activate_last := ACTIVATE; (* letzten Status sichern zur Flankenerkennung *)

(* IP_FIFO *)
IP_FIFO(FIFO:=IP_C.FIFO,STATE:=ip_state,ID:=ip_id);

(* revision history
ks	18. oct. 2008	rev 1.0
	original version

ks	20. oct. 2009	rev 1.1
	Networkbuffer und Buffer-funktionen auf Basis 0

*)

(***************************************************************************************)
(*               SNTP Datenstruktur
                                  1                   2                   3   
              0 1 2 3 4 5 6 7 8 9 0 1 2 3 4 5 6 7 8 9 0 1 2 3 4 5 6 7 8 9 0 1 
             +-+-+-+-+-+-+-+-+-+-+-+-+-+-+-+-+-+-+-+-+-+-+-+-+-+-+-+-+-+-+-+-+
Byte: 01-04  |LI | VN  |Mode |    Stratum    |     Poll      |   Precision   |
             +-+-+-+-+-+-+-+-+-+-+-+-+-+-+-+-+-+-+-+-+-+-+-+-+-+-+-+-+-+-+-+-+
Byte: 05-08  |                          Root  Delay (32 Bit)                 |
             +-+-+-+-+-+-+-+-+-+-+-+-+-+-+-+-+-+-+-+-+-+-+-+-+-+-+-+-+-+-+-+-+
Byte: 09-12  |                       Root  Dispersion (32 Bit)               |
             +-+-+-+-+-+-+-+-+-+-+-+-+-+-+-+-+-+-+-+-+-+-+-+-+-+-+-+-+-+-+-+-+
Byte: 13-16  |                     Reference Identifier (32 Bit)             |
             +-+-+-+-+-+-+-+-+-+-+-+-+-+-+-+-+-+-+-+-+-+-+-+-+-+-+-+-+-+-+-+-+
Byte: 17-24  |                    Reference Timestamp (64 Bit)               |
             +-+-+-+-+-+-+-+-+-+-+-+-+-+-+-+-+-+-+-+-+-+-+-+-+-+-+-+-+-+-+-+-+
Byte: 25-32  |                    Originate Timestamp (64 Bit)               |
             +-+-+-+-+-+-+-+-+-+-+-+-+-+-+-+-+-+-+-+-+-+-+-+-+-+-+-+-+-+-+-+-+
Byte: 33-40  |                     Receive Timestamp (64 Bit)                |
             +-+-+-+-+-+-+-+-+-+-+-+-+-+-+-+-+-+-+-+-+-+-+-+-+-+-+-+-+-+-+-+-+
Byte: 41-48  |                     Transmit Timestamp (64 Bit)               |
             +-+-+-+-+-+-+-+-+-+-+-+-+-+-+-+-+-+-+-+-+-+-+-+-+-+-+-+-+-+-+-+-+
Byte: 49-52  |                 Key Identifier (optional) (32 Bit)            |
             +-+-+-+-+-+-+-+-+-+-+-+-+-+-+-+-+-+-+-+-+-+-+-+-+-+-+-+-+-+-+-+-+
Byte: 53-68  |                 Message Digest (optional) (128 Bit)           |
             +-+-+-+-+-+-+-+-+-+-+-+-+-+-+-+-+-+-+-+-+-+-+-+-+-+-+-+-+-+-+-+-+

*)

(*
Worldwide NTP-Server


NIST-Zeitserver
• time-a.nist.gov
129.6.15.28 
NIST, Gaithersburg, Maryland 
• time-a.nist.gov
129.6.15.28 
NIST, Gaithersburg, Maryland 
• time-a.timefreq.bldrdoc.gov
132.163.4.101 (Stand: 1. Dezember 1999)
NIST, Boulder, Colorado 
• time-b.timefreq.bldrdoc.gov
132.163.4.102 (Stand: 1. Dezember 1999)
NIST, Boulder, Colorado 
• time-c.timefreq.bldrdoc.gov
132.163.4.103 (Stand: 1. Dezember 1999)
NIST, Boulder, Colorado 
• utcnist.colorado.edu
128.138.140.44
University of Colorado, Boulder 
• time.nist.gov
192.43.244.18
NCAR, Boulder, Colorado 
• time-nw.nist.gov
131.107.1.10
Microsoft, Redmond, Washington 
• nist1.dc.certifiedtime.com
216.200.93.8
Abovnet, North Virginia 
• nist1.datum.com
209.0.72.7
Datum, San Jose, Kalifornien 
• nist1.nyc.certifiedtime.com
208.184.49.129 
Abovnet, New York City 
• nist1.sjc.certifiedtime.com
207.126.103.202
Abovnet, San Jose, Kalifornien 

Zeitserver der ersten Ebene
Sortiert nach Standort: 
Nordamerika
• Palo Alto, Kalifornien: Systems Research Center, Compaq Computer Corp.
204.123.2.72: usno.pa-x.dec.com; CNAME: navobs1.pa-x.dec.com
Servicebereich: US-Zeitzonen PST (Pacific Standard Time) und MST (Mountain Standard Time) 
• Marina del Rey, Kalifornien: USC Information Sciences Institute
128.9.176.30: timekeeper.isi.edu
Servicebereich: CalRen2- und Los Nettos-Bereich  
• Washington, DC: U.S. Naval Observatory
192.5.41.41: tock.usno.navy.mil 
192.5.41.40: tick.usno.navy.mil
Servicebereich: NSFNET 
• Ottawa, Ontario, Kanada: National Research Council of Canada
time.chu.nrc.ca
Servicebereich: Kanada 
• Raleigh, North Carolina: North Carolina State University
152.1.58.124: terrapin.csc.ncsu.edu
Servicebereich: Südosten der USA 
• Cambridge, Massachusetts: MIT Information Systems
18.72.0.3: bitsy.mit.edu 
Servicebereich: NSFNET- und NEARnet-Bereich 
• Cambridge, Massachusetts: MIT
18.26.4.105: bonehed.lcs.mit.edu
Servicebereich: Osten der USA 
• Palo Alto, Kalifornien: Internet Software Consortium
192.5.5.250: clock.isc.org
Servicebereich: BARRnet, Alternet-West und CIX-West 
• Cambridge, Massachusetts: Open Software Foundation
130.105.4.59: clock.osf.org
Servicebereich: NSFNET- und NEARnet-Bereich 
• Palo Alto, Kalifornien: ViaNet Communications
209.81.9.7: clock.via.net 
• Cleveland, Ohio: Lewis Research Center (NASA)
128.156.1.43: lerc-dns.lerc.nasa.gov
Servicebereich: NSFNET und OARNET 
• Colorado Springs, Colorado: Schriever AFB
204.34.198.40: navobs1.usnogps.navy.mil; CNAME: tick.usnogps.navy.mil 
204.34.198.41: navobs1.usnogps.navy.mil; CNAME: tock.usnogps.navy.mil 
Servicebereich: US-Zeitzonen PST (Pacific Standard Time) und MST (Mountain Standard Time) 
• St. Louis, Missouri: Washington University
128.252.19.1: navobs1.usnogps.navy.mil; CNAME: tick.wustl.edu 
Servicebereich: US-Zeitzone CST (Central Standard Time) 
• Research Triangle Park, North Carolina: MCNC
192.101.21.1: ncnoc.ncren.net
Servicebereich: NC-REN-Bereich (North Carolina Research and Education Network) 
• Cupertino, Kalifornien: HP
192.6.38.127: ntp-cup.external.hp.com
Servicebereich: USA Westküste 
• Newark, Delaware: Conectiv Communications
138.39.7.20: ntp1.delmarva.com
Servicebereich: Cable & Wireless Network (früher MCInet) 
• University Park, Pennsylvania: Penn State University
128.118.46.3: otc1.psu.edu
Servicebereich: NSFNET, PREPNET und JvNCnet  

Europa
• Borowiec, Polen: Astrogeodynamical Observatory, Space Research Centre
150.254.183.15: vega.cbk.poznan.pl
Servicebereich: Polen und Europa 
• Stockholm, Schweden: Stupi AB
192.36.143.151: Time2.Stupi.SE
Servicebereich: Europa 
• Turin, Italien: IEN Galileo Ferraris
193.204.114.1: time.ien.it
Servicebereich: Italien und Europa 
• Zürich, Schweiz: Integrated Systems Laboratory , Eidgenössischen Technischen Hochschule Zürich 
129.132.2.21: swisstime.ethz.ch
Servicebereich: Schweiz und Europa 
• Turin, Italien: CSTV of National Research Council
150.145.33.1: tempo.cstv.to.cnr.it
Servicebereich: Italien und Europa 
• Erlangen, Deutschland: Universität Erlangen-Nürnberg
ntp0.fau.de; ntp1.fau.de; ntp2.fau.de; 
ntps1-0.uni-erlangen.de; ntps1-1.uni-erlangen.de; ntps1-2.uni-erlangen.de
Servicebereich: Deutschland und Europa 
• Berlin, Deutschland: Technische Universität Berlin
130.149.17.21: ntps1-0.cs.tu-berlin.de
130.149.17.8: ntps1-1.cs.tu-berlin.de
Servicebereich: Deutschland und Europa 
• Deutschland
131.173.17.7: ntps1-1.rz.Uni-Osnabrueck.DE
Servicebereich: Deutschland und Europa 
• Schweden
192.36.143.150: Time1.Stupi.SE
Servicebereich: SUnet und NORDUnet Schweden 

Fernost und pazifische Randgebiete
• Hong Kong: Chinesische Universität von Hong Kong. 
137.189.6.18: clock.cuhk.edu.hk
Servicebereich: Hong Kong (China) und Südostasien  
• Fukuoka, Japan: Universität Fukuoka
133.100.9.2: clock.nc.fukuoka-u.ac.jp
133.100.11.8: clock.tl.fukuoka-u.ac.jp
Servicebereich: Japan und pazifischer Raum  

Australien
• Melbourne, Australien: University of Melbourne
128.250.36.2: ntp.cs.mu.OZ.AU
Servicebereich: Australien und Neuseeland  

Zeitserver der zweiten Ebene
Nach geographischem Standort sortiert: 
Nordamerika
NTP-Zeitserver: • Quebec, Kanada: Canadian Meteorological Center
ntp1.cmc.ec.gc.ca; ntp2.cmc.ec.gc.ca 
Servicebereich: Ostkanada  
• Ontario, Kanada: National Research Council of Canada
time.chu.nrc.ca; time.nrc.ca
Servicebereich: Kanada 
• Saskatchewan, Kanada: University of Regina 
142.3.100.15: timelord.uregina.ca
Servicebereich: Kanada 
• Ontario, Kanada: University of Toronto
tick.utoronto.ca; tock.utoronto.ca
Servicebereich: Ostkanada  
• Mexiko: Audiotel-Büro 
ntp2a.audiotel.com.mx; ntp2c.audiotel.com.mx; ntp2b.audiotel.com.mx
Servicebereich: Avantel, MCINet und Mexiko 
• Santa Cruz, Kalifornien: Scruz-net, inc.
165.227.1.1: ns.scruz.net
Servicebereich: Westen der USA 
• San Diego, Kalifornien: UCSD Academic Computing Services/Network Operations
132.239.254.49: ntp.ucsd.edu
Servicebereich: CERFNET; NSFNET, SDSC-Bereich, und nahegelegene Bereiche 
• Quincy, Kalifornien 
ntp1.mainecoon.com; ntp2.mainecoon.com 
Servicebereich: Nordamerika 
• Newark, Delaware: University of Delaware
128.175.1.3: louie.udel.edu
Servicebereich: CAIRN, Abilene und vBNS  
• Atlanta, Georgia: CNSG
ntp.shorty.com
Servicebereich: Südwesten der USA  
• Kennesaw, Georgia: PeachNet 
rolex.peachnet.edu; timex.peachnet.edu
Servicebereich: PeachNet (Georgia) und Südwesten der USA  
• Urbana-Champaign, Illinois: University of Illinois
ntp-0.cso.uiuc.edu; ntp-1.cso.uiuc.edu; ntp-2.cso.uiuc.edu
Servicebereich: CICNET, Mittlerer Westen und NCSA-Bereich  
• Chicago, Illinois: Argonne National Laboratory 
ntp-1.mcs.anl.gov; ntp-2.mcs.anl.gov
Servicebereich: NSF/ANSNet, CICNet, NetIllinois und ESNet  
• West Lafayette, Indiana: Purdue University
gilbreth.ecn.purdue.edu; harbor.ecn.purdue.edu; molecule.ecn.purdue.edu 
Servicebereich: NSFNET- und CICNET-Bereich  
• Manhattan, Kansas: KansasNet OnLine Services
199.240.130.1: ntp1.kansas.net
199.240.130.12: ntp2.kansas.net
Servicebereich: Zentral-USA und Great Plains  
• Boston, Massachusetts: UMass-Boston CS dept.
158.121.104.4: timeserver.cs.umb.edu
Servicebereich: Neuengland  
• Minneapolis/St Paul, Minnesota: University of Minnesota
ns.nts.umn.edu; nss.nts.umn.edu
Servicebereich: CICNET-Bereich  
• Columbia, Missouri: University of Missouri-Columbia
128.206.206.12: everest.cclabs.missouri.edu
Servicebereich: MOREnet  
• Omaha, Nebraska: Radiks Internet Access
205.138.126.83: allison.radiks.net
Servicebereich: Mittlerer Westen, USA  
• Las Vegas, Nevada: University of Nevada System Computing Services
131.216.1.101: cuckoo.nevada.edu 
Servicebereich: NevadaNet, NSFNET und SDSC-Bereich  
• Las Vegas, Nevada: UNLV College of Engineering
tick.cs.unlv.edu; tock.cs.unlv.edu
Servicebereich: Sprintnet  
• New York City, New York: Columbia University
ntp.ctr.columbia.edu 
Servicebereich: Sprintlink und NYSERnet  
• Ithaca, New York: Cornell University 
192.35.82.50: ntp0.cornell.edu
Servicebereich: NSFNET und NYSER-Bereich  
• New York, New York: Morningside Campus, Columbia University
sundial.columbia.edu
Servicebereich: NYSERnet  
• New York City, New York: Columbia University Computer Science Department
timex.cs.columbia.edu 
Servicebereich: PSINET; NSFNET, und NYSER-Bereich  
• Norman, Oklahoma: University of Oklahoma
129.15.22.8: constellation.ecn.uoknor.edu 
Servicebereich: Midnet  
• Coos Bay, Oregon: Koala Computers
207.48.109.6: tick.koalas.com
Servicebereich: Nordwesten der USA  
• University Park, Pennsylvania: Penn State University
128.118.25.3: clock.psu.edu
Servicebereich: Internet2, vBNS, CERFnet(AT&T IP Services), PSC/NCNE und CASC 
• Pittsburgh, Pennsylvania: Pittsburgh Supercomputing Center
128.182.58.100: fuzz.psc.edu
Servicebereich: NSFNET und PSC-Bereich  
• Pittsburgh, Pennsylvania: Carnegie Mellon Electrical and Computer Engineering 
ntp-1.ece.cmu.edu; ntp-2.ece.cmu.edu 
Servicebereich: PREPNET und PSC-Bereich  
• Dallas, Texas: Cox School of Business, Southern Methodist University
129.119.80.126: ntp.cox.smu.edu 
Servicebereich: NSFNET und SESQUI-Bereich  
• Hughes Springs, Texas: First National Bank
209.144.20.76: ntp.fnbhs.com
Servicebereich: Nordosten Texas  
• Houston, Texas: Baylor College of Medicine
128.249.1.10: ntp.tmc.edu 
Servicebereich: NSFNET und SESQUI-Bereich  
• College Station, Texas: Texas A&M University
165.91.52.110: ntp5.tamu.edu
Servicebereich: NSFNET, SESQUI-Bereich, THEnet und TAMUSDSN 
• Plano, Texas: Greyware Automation Products
tick.greyware.com; tock.greyware.com
Servicebereich: Südzentral-USA  
• Blacksburg, Virginia: Virginia Tech Computing Center
ntp-1.vt.edu; ntp-2.vt.edu
Servicebereich: Südwesten der USA  
• Arlington, Virginia: Center for Seismic Studies
140.162.1.3: ntp.cmr.gov
Servicebereich: NSFNET und SURA-Bereich  
• Richland, Washington: Washington State University 
192.31.216.30: clock.tricity.wsu.edu
Servicebereich: NSFNET und NorthWestNet  
• Washington, USA: Mill Creek
time.ultimeth.net
Servicebereich: Nordwesten der USA  
• Wisconsin, USA: Computer Science Department, University of Wisconsin-Madison
ntp1.cs.wisc.edu; ntp2.cs.wisc.edu; ntp3.cs.wisc.edu
Servicebereich: USA und jeder andere  

Südamerika
• Buenos Aires, Argentinien: Network Access Point
200.49.40.1: CNAME: tick.nap.com.ar
200.49.32.1: CNAME: tock.nap.com.ar
Servicebereich: Argentinien 
• Buenos Aires, Argentinien: Sinectis S.A.
time.sinectis.com.ar 
Servicebereich: Argentinien 
• Brasilien: Brazilian Research Network
200.144.121.33: ntp.cais.rnp.br 
Servicebereich: Brasilien 
• Venezuela: VELUG, Grupo de Usuarios Linux de Venezuela
150.185.192.250: ntp.linux.org.ve
Servicebereich: Arica  

Europa
• Zürich, Schweiz: Eidgenössischen Technischen Hochschule Zürich
129.132.98.11: bernina.ethz.ch
Servicebereich: Schweiz und Europa  
• Standort: Kopenhagen, Dänemark, Europa 
clock.netcetera.dk; clock2.netcetera.dk 
Servicebereich: Dänemark, Skandinavien und Nordeuropa  
• Spanien: Altea 
slug.ctv.es
Servicebereich: Spanien  
• Pieksamaki, Finnland: Keski-Savon Oppimiskeskus
tick.keso.fi; tock.keso.fi
Servicebereich: Finnland  
• Meudon, Frankreich: Observatoire de Paris-Meudon 
ntp.obspm.fr 
Servicebereich: Frankreich und Europa  
• Lyon, Frankreich: CISM 
ntp.univ-lyon1.fr 
Servicebereich: Frankreich, Schweiz, Italien und Europa  
• Paris, Frankreich: VIA, Ecole Centrale
138.195.130.70: ntp.via.ecp.fr
Servicebereich: Frankreich und Europa  
• Budapest, Ungarn: KFKI Research Institute for Particle and Nuclear Physics
148.6.0.1: time.kfki.hu
Servicebereich: HUNGARNET  
• Italien: Net4u Srl, Vercelli, Italien
195.32.52.129: ntps.net4u.it
Servicebereich: Italien  
• Oslo, Norwegen: Universität Oslo
129.240.64.3: fartein.ifi.uio.no 
Servicebereich: NORDUnet  
• Oslo, Norwegen: Alcanet International
time.alcanet.no
Servicebereich: Europa 
• Krakau, Polen: Academic Computer Centre 
149.156.4.11: info.cyf-kr.edu.pl
Servicebereich: Polen und Europa  
• Lund, Schweden: Lund Institute of Technology
130.235.20.3: ntp.lth.se 
Servicebereich: Schweden und NORDUnet 
• Ljubljana, Slowenien: Institute of Biophysics, University of Ljubljana
biofiz.mf.uni-lj.si 193.2.69.11
Servicebereich: Slowenien und Europa  
• Ljubljana, Slowenien: Hydrometeorological Institute of Slovenia
hmljhp.rzs-hm.si
Servicebereich: Slowenien und Europa  
• Ljubljana, Slowenien: Academic and Research Network of Slovenia
ntp1.arnes.si; ntp2.arnes.si
Servicebereich: Slowenien und Europa  
• Ljubljana, Slowenien: J. Stefan Institute
time.ijs.si
Servicebereich: Slowenien und Europa  

Britische Inseln
• Dublin, Irland: School of Mathematics, Trinity College 
ntp.cs.tcd.ie; ntp.maths.tcd.ie; ntp.tcd.ie
Servicebereich: Irland und Großbritannien 
• Glasgow, Schottland: Strathclyde University 
ntp.cs.strath.ac.uk 
Servicebereich: Großbritannien, Europa und andere 
• Cambridge, Großbritannien
ntp0.uk.uu.net; ntp1.uk.uu.net; 
ntp2.uk.uu.net 
Servicebereich: UUNET (in Großbritannien früher auch als PIPEX bekannt) und Großbritannien.  
• Manchester, England: University of Manchester
ntp2a.mcc.ac.uk; ntp2b.mcc.ac.uk;
ntp2c.mcc.ac.uk; ntp2d.mcc.ac.uk 
Servicebereich: Großbritannien  
• Buckinghamshire, Großbritannien: Wibble U.K., Aylesbury
tick.tanac.net
Servicebereich: Großbritannien  

Asien
• Moskau, Russland: Landau Institute for Theoretical Physics
193.233.9.7: ntp.landau.ac.ru
Servicebereich: Russland  
• Russland: Pushchino (bei Moskau)
194.149.67.130: ntp.psn.ru
Servicebereich: Russland 
• Chernogolovka, Russland: Chernogolovka Scientific Center (bei Moskau)
193.233.46.10: sign.chg.ru
Servicebereich: Russland  

Fernost und pazifische Randgebiete
• Tokyo, Japan: Cyber Fleet, Inc.
203.139.30.195: ntp.cyber-fleet.net
Servicebereich: Japan und Ostasien  
• Seoul, Korea: Inet, Inc.
time.nuri.net
Servicebereich: Korea, Japan, Hong Kong und Ostasien  
• Hamilton, Neuseeland: Universität Waikato
truechimer.waikato.ac.nz; truechimer1.waikato.ac.nz; 
truechimer2.waikato.ac.nz; truechimer3.waikato.ac.nz
Servicebereich: Neuseeland  
• Singapur und Philippinen: 
ntp.shim.org 
Servicebereich: Singapur  

Afrika
• Lagos, Nigeria: Supernet300
ntp.supernet300.com
Servicebereich: Westafrika (hauptsächlich nigerischer NITEL-Backbone)  
• Pietermaritzburg, Südafrika: Natal University
143.128.82.200: ntp.cs.unp.ac.za
Servicebereich: Südafrika  

Australien
• Adelaide, Südaustralien: University of Adelaide
129.127.28.4: augean.eleceng.adelaide.edu.au
129.127.40.3: ntp.adelaide.edu.au
203.21.37.18: ntp.saard.net
Servicebereich: AARNet  
• Carlton, Victoria, Australien: eSec Limited
203.21.84.4: time.esec.com.au  

*)
END_FUNCTION_BLOCK

(* POU SNTP_SERVER, ST *)
FUNCTION_BLOCK SNTP_SERVER
VAR_IN_OUT
	IP_C : IP_C; (* IP_Control Verwaltungsstruktur *)
	S_BUF : NETWORK_BUFFER;
	R_BUF : NETWORK_BUFFER;
END_VAR
VAR_INPUT
	ENABLE : BOOL;
	STRATUM : BYTE := BYTE#1;
	UDT : DT;
	XMS : INT;
END_VAR
VAR
	IP_FIFO : IP_FIFO;
	ip_state : BYTE;
	ip_id : BYTE;
	i2 : INT;
	i : INT;
	timestamp_int : DWORD; (* Timestamp integer part *)
	timestamp_sek : DWORD; (* Timestamp fraction part (HIGH_WORD) *)
	ts_b : BYTE;
	state : INT;
	tx : UDINT;
END_VAR

(*
	version 1.1		20. oct. 2009
	programmer 		ks
	tested BY		ks

	SNTP_SERVER stellt Datum/Uhrzeit füR andere (S)NTP_CLIENTS zur Verfügung.
*)
(* Domain Name System (query) *)
tx := T_PLC_MS(); (* read system time *)

CASE state OF

00: (* Warten auf Freigabe *)
	IF ENABLE THEN
		state := 10;
		ip_state := BYTE#1; (* Anmelden *)
	END_IF;

10: (* Bei IP_Control anmelden und auf freigabe warten *)
	IF ip_state = BYTE#3 THEN
		(* IP Datenverkehr einrichten *)
		IP_C.C_PORT := WORD#123; (* Portnummer eintragen *)
		IP_C.C_IP := DWORD#00; (* IP eintragen *)
		IP_C.C_MODE := BYTE#5; (* Mode: UDP+PASSIV+PORT *)
		IP_C.C_ENABLE := TRUE; (* Verbindungsaufbau freigeben *)
		IP_C.TIME_RESET := TRUE; (* Zeitueberwachung rücksetzen *)
		IP_C.R_OBSERVE := FALSE; (* Datenempfang ueberwachen *)
		S_BUF.SIZE := UINT#0; (* Sendelänge eintragen *)
		R_BUF.SIZE := UINT#0; (* Empfangslänge rücksetzen *)
		state := 20;
	END_IF;
20:
	IF R_BUF.SIZE > UINT#0 THEN
		state := 20;
		(* empfangenes Telegramm mit 00 auffüllen , wenn zu kurz ! und Sendebuffer mit 00 vorbelegen *)
		FOR i := 0 TO 47 DO
			IF INT_TO_UINT(i) > R_BUF.SIZE - 1 THEN
				R_BUF.BUFFER[i] := BYTE#00;
			END_IF;
			S_BUF.BUFFER[i] := BYTE#00;
		END_FOR;

		R_BUF.SIZE := UINT#0;

		(* Sendedaten aufbereiten *)
		S_BUF.BUFFER[0] := BYTE#2#11100; (* Flags: NO WARNING, NTP VERSION 3 , SERVER *)
		S_BUF.BUFFER[1] := STRATUM; (* Peer Clock Stratum: *)
		S_BUF.BUFFER[2] := BYTE#10; (* Peer Polling Intervall 2 hoch 10 = 1024 sek. *)
		S_BUF.BUFFER[3] := BYTE#16#FB; (* Peer Clock Precision: -5 = -31,25ms *)

		(* Umrechnung SNTP Timestamp Base 1900-01-01 = Unix 1970-01-01 + 2208988800 sekunden *)
		timestamp_int := DT_TO_DWORD(UDT) + DWORD#2208988800;

		(* Sekundenanteile sind als 32 Bit Fractal dargestellt *)
		(* nur mit veringerte Auflösung berechnen 1/65535 -> Highword verwenden *)
		(* Berechnung des Sekundenanteils: xms * 65535 / 1000 *)
		timestamp_sek := DINT_TO_DWORD(DWORD_TO_DINT(SHL(INT_TO_DWORD(XMS),16))/DINT#1000);

		ts_b := BYTE_OF_DWORD(timestamp_int,3); (* Timestamp Byte 3 *)
		S_BUF.BUFFER[16] := ts_b; (* Reference Timestamp *)
		S_BUF.BUFFER[32] := ts_b; (* Receive   Timestamp *)
		S_BUF.BUFFER[40] := ts_b; (* Transmit  Timestamp *)

		ts_b := BYTE_OF_DWORD(TIMESTAMP_INT,2); (* Timestamp Byte 2 *)
		S_BUF.BUFFER[17] := ts_b; (* Reference Timestamp *)
		S_BUF.BUFFER[33] := ts_b; (* Receive   Timestamp *)
		S_BUF.BUFFER[41] := ts_b; (* Transmit  Timestamp *)

		ts_b := BYTE_OF_DWORD(TIMESTAMP_INT,1); (* Timestamp Byte 1 *)
		S_BUF.BUFFER[18] := ts_b; (* Reference Timestamp *)
		S_BUF.BUFFER[34] := ts_b; (* Receive   Timestamp *)
		S_BUF.BUFFER[42] := ts_b; (* Transmit  Timestamp *)

		ts_b := BYTE_OF_DWORD(TIMESTAMP_INT,0); (* Timestamp Byte 0 *)
		S_BUF.BUFFER[19] := ts_b; (* Reference Timestamp *)
		S_BUF.BUFFER[35] := ts_b; (* Receive   Timestamp *)
		S_BUF.BUFFER[43] := ts_b; (* Transmit  Timestamp *)

		ts_b := BYTE_OF_DWORD(TIMESTAMP_SEK,1); (* Timestamp Byte 1 *)
		S_BUF.BUFFER[20] := ts_b; (* Reference Timestamp *)
		S_BUF.BUFFER[36] := ts_b; (* Receive   Timestamp *)
		S_BUF.BUFFER[44] := ts_b; (* Transmit  Timestamp *)

		ts_b := BYTE_OF_DWORD(timestamp_sek,0);	(* Timestamp Byte 0 *)
		S_BUF.BUFFER[21] := ts_b; (* Reference Timestamp *)
		S_BUF.BUFFER[37] := ts_b; (* Receive   Timestamp *)
		S_BUF.BUFFER[45] := ts_b; (* Transmit  Timestamp *)

		(* Byte 1-8 von Transmit-Time auf Originate-Time umkopieren *)
		i2 := 40;
		FOR i := 24 TO 31 DO
			S_BUF.BUFFER[i] := R_BUF.BUFFER[i2];
			i2 := i2 +1;
		END_FOR;

		S_BUF.SIZE := UINT#48; (* Daten senden *)

	ELSIF NOT ENABLE AND S_BUF.SIZE = UINT#0 THEN
		ip_state := BYTE#4; (* Abmelden *)
		state := 0;
	END_IF;

END_CASE;

(* IP_FIFO *)
IP_FIFO(FIFO:=IP_C.FIFO,STATE:=ip_state,ID:=ip_id);

(* revision history
ks	18. oct. 2008	rev 1.0
	original version

ks	20. oct. 2009	rev 1.1
	Networkbuffer und Buffer-funktionen auf Basis 0

*)


(*               SNTP(NTP) Datenstruktur
                                  1                   2                   3
              0 1 2 3 4 5 6 7 8 9 0 1 2 3 4 5 6 7 8 9 0 1 2 3 4 5 6 7 8 9 0 1
             +-+-+-+-+-+-+-+-+-+-+-+-+-+-+-+-+-+-+-+-+-+-+-+-+-+-+-+-+-+-+-+-+
Byte: 01-04  |LI | VN  |Mode |    Stratum    |     Poll      |   Precision   |
             +-+-+-+-+-+-+-+-+-+-+-+-+-+-+-+-+-+-+-+-+-+-+-+-+-+-+-+-+-+-+-+-+
Byte: 05-08  |                          Root  Delay (32 Bit)                 |
             +-+-+-+-+-+-+-+-+-+-+-+-+-+-+-+-+-+-+-+-+-+-+-+-+-+-+-+-+-+-+-+-+
Byte: 09-12  |                       Root  Dispersion (32 Bit)               |
             +-+-+-+-+-+-+-+-+-+-+-+-+-+-+-+-+-+-+-+-+-+-+-+-+-+-+-+-+-+-+-+-+
Byte: 13-16  |                     Reference Identifier (32 Bit)             |
             +-+-+-+-+-+-+-+-+-+-+-+-+-+-+-+-+-+-+-+-+-+-+-+-+-+-+-+-+-+-+-+-+
Byte: 17-24  |                    Reference Timestamp (64 Bit)               |
             +-+-+-+-+-+-+-+-+-+-+-+-+-+-+-+-+-+-+-+-+-+-+-+-+-+-+-+-+-+-+-+-+
Byte: 25-32  |                    Originate Timestamp (64 Bit)               |
             +-+-+-+-+-+-+-+-+-+-+-+-+-+-+-+-+-+-+-+-+-+-+-+-+-+-+-+-+-+-+-+-+
Byte: 33-40  |                     Receive Timestamp (64 Bit)                |
             +-+-+-+-+-+-+-+-+-+-+-+-+-+-+-+-+-+-+-+-+-+-+-+-+-+-+-+-+-+-+-+-+
Byte: 41-48  |                     Transmit Timestamp (64 Bit)               |
             +-+-+-+-+-+-+-+-+-+-+-+-+-+-+-+-+-+-+-+-+-+-+-+-+-+-+-+-+-+-+-+-+
Byte: 49-52  |                 Key Identifier (optional) (32 Bit)            |
             +-+-+-+-+-+-+-+-+-+-+-+-+-+-+-+-+-+-+-+-+-+-+-+-+-+-+-+-+-+-+-+-+
Byte: 53-68  |                 Message Digest (optional) (128 Bit)           |
             +-+-+-+-+-+-+-+-+-+-+-+-+-+-+-+-+-+-+-+-+-+-+-+-+-+-+-+-+-+-+-+-+
*)
END_FUNCTION_BLOCK

(* POU SYS_LOG, ST *)
FUNCTION_BLOCK SYS_LOG
VAR_IN_OUT
	IP_C : IP_C; (* IP_Control Verwaltungsstruktur *)
	S_BUF : NETWORK_BUFFER;
	R_BUF : NETWORK_BUFFER;
END_VAR
VAR_INPUT
	ACTIVATE : BOOL;
	LDT : DT;
	SERVER_IP4 : DWORD;
	PORT : WORD;
	FACILITY : BYTE;
	SEVERITY : BYTE;
	TAG : STRING(32);
	HOSTNAME : STRING;
	MESSAGE : STRING(STRING_LENGTH);
	OPTION : BYTE;
END_VAR
VAR_OUTPUT
	DONE_P : BOOL;
	ERROR : DWORD;
END_VAR
VAR
	ip_state : BYTE;
	ip_id : BYTE;
	IP_FIFO : IP_FIFO;
	activate_last : BOOL;
	state : INT;
	s1 : STRING(20);
	i : INT;
END_VAR

(*
version 1.1		20. jun. 2009
programmer 		ks
tested by		ks

SYSLOG versendet Meldungen auf Basis des SYSLOG-Standards

*)
CASE state OF
00: (* auf positive Flanke SET warten *)
	IF ACTIVATE AND NOT ACTIVATE_LAST THEN
		state := 10;
		ERROR := DWORD#0;
		IP_STATE := BYTE#1; (* Anmelden *)
	END_IF;
	DONE_P := FALSE;

10: (* Bei IP_Control anmelden und auf freigabe warten *)
	IF IP_STATE = BYTE#3 THEN
		(* Sendedaten aufbereiten *)
		i := 0;
		IF (OPTION AND BYTE#0000_0001) = BYTE#00 THEN (* Option: no priority Code *)
			(* Priority:  '<xx>' als dezimalwert *)
			(* BYTE: xxxx x...  = Facility *)
			(*       .... .xxx  = Level *)
			s1 := REPLACE('<P>',BYTE_TO_STRING(SHL(FACILITY,3) OR (SEVERITY AND BYTE#0000_0111)),1,2);
		ELSE
			s1 := '';
		END_IF;

		IF (OPTION AND BYTE#0000_0010) = BYTE#00 THEN (* Option: No Use Syslog RFC Header *)
			(* 'month day hh:mm:ss ' *)
			s1 := CONCAT(s1,DT_TO_STRF(DTI:=LDT,MS:=0,FMT:='#E #W #N:#R:#T ',LANG:=1));
			_STRING_TO_BUFFER(STR:=s1,POS:=i,PT:=ADR(S_BUF.BUFFER),SIZE:=UINT#1024);
			i := i + LEN(s1);
			(* ' sourcename eintragen *)
			_STRING_TO_BUFFER(STR:=HOSTNAME,POS:=i,PT:=ADR(S_BUF.BUFFER),SIZE:=UINT#1024);
			i := i + LEN(HOSTNAME);
			S_BUF.BUFFER[i] := BYTE#32; (* leerzeichen einfuegen *)
			i := i + 1;
			(* ' tag eintragen *)
			_STRING_TO_BUFFER(STR:=TAG,POS:=i,PT:=ADR(S_BUF.BUFFER),SIZE:=UINT#1024);
			i := i + LEN(TAG);
			S_BUF.BUFFER[i] := BYTE#32; (* leerzeichen einfuegen *)
			i := i + 1;
		END_IF;

		(* ' message eintragen *)
		_STRING_TO_BUFFER(STR:=MESSAGE,POS:=i,PT:=ADR(S_BUF.BUFFER),SIZE:=UINT#1024);
		i := i + LEN(MESSAGE);

		IF (OPTION AND BYTE#0000_0100) > BYTE#00 THEN (* Option: Add a CR & LF to end of message *)
			S_BUF.BUFFER[i] := BYTE#13; (* Carriage Return einfuegen *)
			i := i + 1;
			S_BUF.BUFFER[i] := BYTE#10; (* Linefeed einfuegen *)
			i := i + 1;
		END_IF;

		state := 30;

		(* IP Datenverkehr einrichten *)
		IF (OPTION AND BYTE#2#0000_1000) > BYTE#00 THEN (* Option: TCP Mode *)
			IP_C.C_MODE := BYTE#0; (* Mode: TCP/AKTIV *)
		ELSE
			IP_C.C_MODE := BYTE#1; (* Mode: UDP/AKTIV *)
		END_IF;

		IF PORT = WORD#0 THEN (* keine Portnummer vorgegeben ? *)
			IF IP_C.C_MODE = BYTE#0 THEN (* Modus bestimmen  TCP oder UDP ? *)
				IP_C.C_PORT := WORD#1468; (* Standard Portnummer für Syslog over TCP *)
			ELSE
				IP_C.C_PORT := WORD#514; (* Standard Portnummer für Syslog over UDP *)
			END_IF;
		ELSE
			IP_C.C_PORT := PORT; (* uebergebene Portnummer eintragen *)
		END_IF;

		IP_C.C_IP := SERVER_IP4; (* IP eintragen *)
		IP_C.C_ENABLE := TRUE; (* Verbindungsaufbau freigeben *)
		IP_C.TIME_RESET := TRUE; (* Zeitueberwachung rücksetzen *)
		IP_C.R_OBSERVE := FALSE; (* Datenempfang ueberwachen *)
		S_BUF.SIZE := INT_TO_UINT(i); (* Sendelänge eintragen *)
		R_BUF.SIZE := UINT#0; (* Empfangslänge rücksetzen *)

	END_IF;

30:
	IF IP_C.ERROR <> DWORD#00 THEN
		ERROR := IP_C.ERROR;
		state := 0;
	ELSIF S_BUF.SIZE = UINT#0 THEN (* warten bis alle daten gesendet sind *)
		DONE_P := TRUE;
		state := 0;
	END_IF;

	IF state = 0 THEN (* Verbindung freigeben *)
		IP_STATE := BYTE#4;
	END_IF;

END_CASE;

ACTIVATE_LAST := ACTIVATE; (* letzten Status sichern zur Flankenerkennung *)

(* IP_FIFO *)
IP_FIFO(FIFO:=IP_C.FIFO,STATE:=ip_state,ID:=IP_ID);

(* revision history
ks	18. oct. 2008	rev 1.0
	original version

ks	20. jun. 2009	rev 1.1
	Networkbuffer und Buffer-funktionen auf Basis 0

*)
END_FUNCTION_BLOCK

(* POU FILE_BLOCK_DEMO, CFC *)
PROGRAM FILE_BLOCK_DEMO
VAR
	PT : NETWORK_BUFFER;
	fsd : FILE_SERVER_DATA;
	FILE_SERVER : FILE_SERVER;
	FILE_BLOCK : FILE_BLOCK;
	filename : STRING := 'config.ini';
	data : BYTE;
	error : BYTE;
	mode : BYTE;
	pos : UDINT;
END_VAR
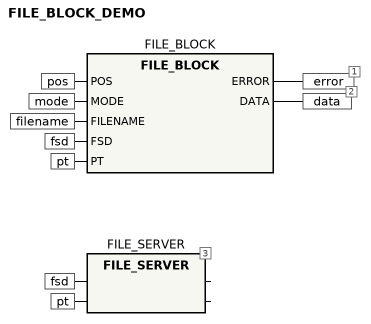
_CFC_ (* Continuous Function Chart, elements in execution order *)
#0 FILE_BLOCK:FILE_BLOCK(POS: pos, MODE: mode, FILENAME: filename, FSD: fsd, PT: pt)
#1 error <= #0.ERROR
#2 data <= #0.DATA
#3 FILE_SERVER:FILE_SERVER(fsd, pt)
_END_CFC_
(* the same logic as Structured Text *)
FILE_BLOCK(POS := pos, MODE := mode, FILENAME := filename, FSD := fsd, PT := pt);
error := FILE_BLOCK.ERROR;
data := FILE_BLOCK.DATA;
FILE_SERVER(fsd, pt);
END_PROGRAM

(* POU FTP_CLIENT_DEMO, CFC *)
PROGRAM FTP_CLIENT_DEMO
VAR
	FTP_CLIENT: FTP_CLIENT;
	ftp_activate: BOOL;
	ftp_done: BOOL;
	ftp_busy: BOOL;
	ftp_error_c: DWORD;
	ftp_error_t: BYTE;
	ftp_url: STRING := 'ftp://581920:123456@oscat.atwebpages.com:2000/subordner/';
	ftp_filename: STRING := 'D:\testfiles\0100kb.bin';
	ftp_download: BOOL := FALSE;
	ftp_activ: BOOL := FALSE;
	file_delete: BOOL := FALSE;
	ftp_timeout: TIME := T#30s;
	zeit : TIME := T#30s;
	stop: BOOL;
	start: BOOL :=TRUE ;
	reset: BOOL;
	error: DWORD;
	ok: DWORD;
	CLK_PRG_1: CLK_PRG;
	COUNT_DR_1: COUNT_DR;
	COUNT_DR_2: COUNT_DR;
END_VAR
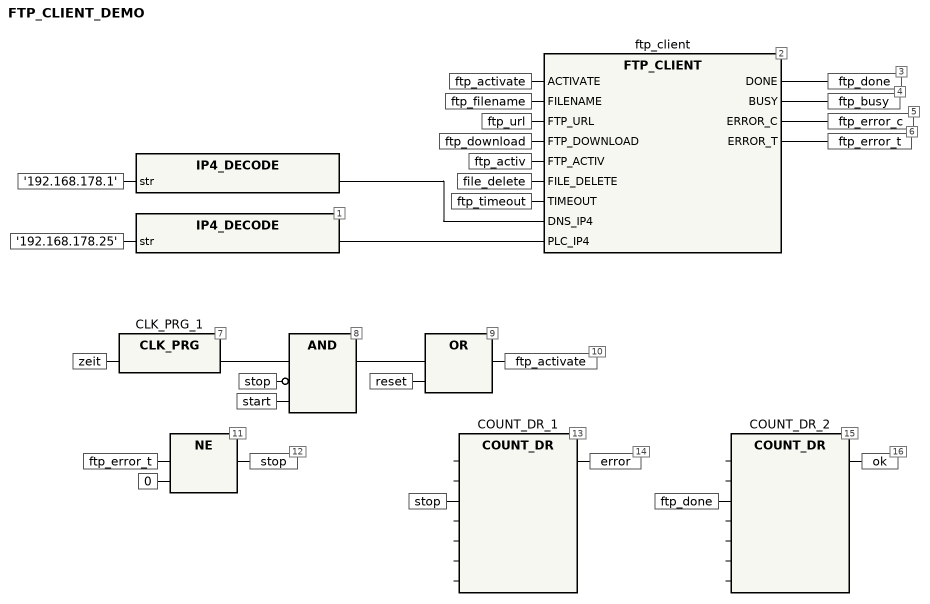
_CFC_ (* Continuous Function Chart, elements in execution order *)
#0 IP4_DECODE(str: '192.168.178.1')
#1 IP4_DECODE(str: '192.168.178.25')
#2 ftp_client:FTP_CLIENT(ACTIVATE: ftp_activate, FILENAME: ftp_filename, FTP_URL: ftp_url, FTP_DOWNLOAD: ftp_download, FTP_ACTIV: ftp_activ, FILE_DELETE: file_delete, TIMEOUT: ftp_timeout, DNS_IP4: #0, PLC_IP4: #1)
#3 ftp_done <= #2.DONE
#4 ftp_busy <= #2.BUSY
#5 ftp_error_c <= #2.ERROR_C
#6 ftp_error_t <= #2.ERROR_T
#7 CLK_PRG_1:CLK_PRG(zeit)
#8 AND(#7, NOT stop, start)
#9 OR(#8, reset)
#10 ftp_activate <= #9
#11 NE(ftp_error_t, 0)
#12 stop <= #11
#13 COUNT_DR_1:COUNT_DR(-, -, stop, -, -, -, -)
#14 error <= #13
#15 COUNT_DR_2:COUNT_DR(-, -, ftp_done, -, -, -, -)
#16 ok <= #15
_END_CFC_
END_PROGRAM

(* POU GET_WAN_IP_DEMO, CFC *)
PROGRAM GET_WAN_IP_DEMO
VAR
	GET_WAN_IP: GET_WAN_IP;
	IP_C: IP_C;
	S_BUF: NETWORK_BUFFER;
	R_BUF: NETWORK_BUFFER;
	IP_CONTROL_1: IP_CONTROL;
	activate: BOOL;
	done: BOOL;
	error_c: DWORD;
	error_t: BYTE;
	wan_ip: STRING;
	new_ip: BOOL;
END_VAR
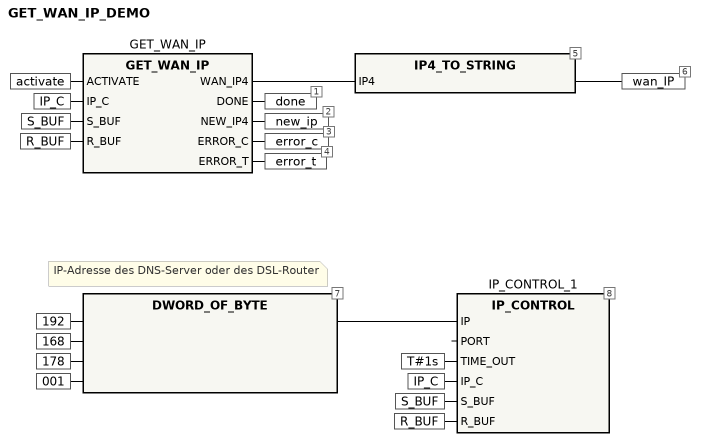
_CFC_ (* Continuous Function Chart, elements in execution order *)
(* IP-Adresse des DNS-Server oder des DSL-Router *)
#0 GET_WAN_IP:GET_WAN_IP(ACTIVATE: activate, IP_C: IP_C, S_BUF: S_BUF, R_BUF: R_BUF)
#1 done <= #0.DONE
#2 new_ip <= #0.NEW_IP4
#3 error_c <= #0.ERROR_C
#4 error_t <= #0.ERROR_T
#5 IP4_TO_STRING(IP4: #0.WAN_IP4)
#6 wan_IP <= #5
#7 DWORD_OF_BYTE(192, 168, 178, 001)
#8 IP_CONTROL_1:IP_CONTROL(IP: #7, PORT: -, TIME_OUT: T#1s, IP_C: IP_C, S_BUF: S_BUF, R_BUF: R_BUF)
_END_CFC_
(* the same logic as Structured Text *)
(* IP-Adresse des DNS-Server oder des DSL-Router *)
GET_WAN_IP(ACTIVATE := activate, IP_C := IP_C, S_BUF := S_BUF, R_BUF := R_BUF);
done := GET_WAN_IP.DONE;
new_ip := GET_WAN_IP.NEW_IP4;
error_c := GET_WAN_IP.ERROR_C;
error_t := GET_WAN_IP.ERROR_T;
wan_IP := IP4_TO_STRING(IP4 := GET_WAN_IP.WAN_IP4);
IP_CONTROL_1(IP := DWORD_OF_BYTE(192, 168, 178, 001), TIME_OUT := T#1s, IP_C := IP_C, S_BUF := S_BUF, R_BUF := R_BUF);
END_PROGRAM

(* POU HTTP_DEMO, CFC *)
PROGRAM HTTP_DEMO
VAR
	url_text : STRING := 'http://weather.yahooapis.com/forecastrss?p=94089&u=c';
	URL_DATA : URL;
	IP_C: IP_C;
	S_BUF: NETWORK_BUFFER;
	R_BUF: NETWORK_BUFFER;
	IP_CONTROL_1: IP_CONTROL;

	DNS_CLIENT: DNS_CLIENT;
	HTTP_GET: HTTP_GET;
	http_release: BOOL;
	enable: BOOL := TRUE;
	http_status: STRING;
	header_start: UINT;
	header_stop: UINT;
	body_start: UINT;
	body_stop: UINT;
	http_get_done: BOOL;
	http_get_error: DWORD;
	COUNT_DR: COUNT_DR;
	cycles: DWORD;
	TON_1: TON;
	F_TRIG: F_TRIG;
END_VAR
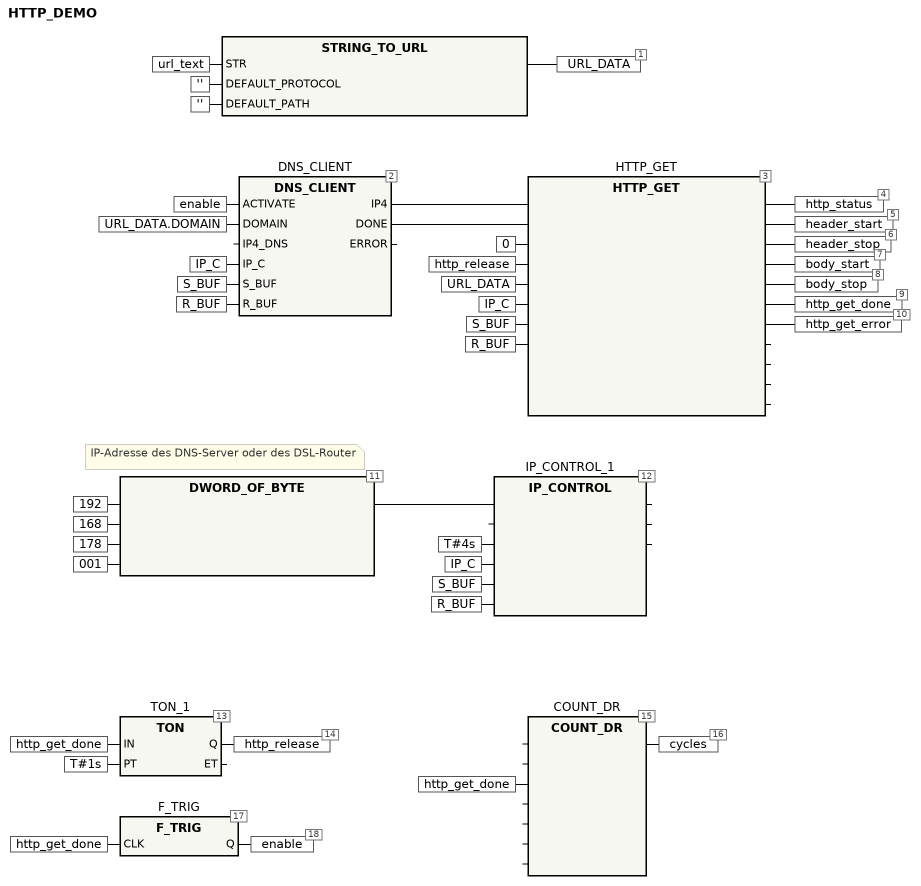
_CFC_ (* Continuous Function Chart, elements in execution order *)
(* IP-Adresse des DNS-Server oder des DSL-Router *)
#0 STRING_TO_URL(STR: url_text, DEFAULT_PROTOCOL: '', DEFAULT_PATH: '')
#1 URL_DATA <= #0
#2 DNS_CLIENT:DNS_CLIENT(ACTIVATE: enable, DOMAIN: URL_DATA.DOMAIN, IP4_DNS: -, IP_C: IP_C, S_BUF: S_BUF, R_BUF: R_BUF)
#3 HTTP_GET:HTTP_GET(#2.IP4, #2.DONE, 0, http_release, URL_DATA, IP_C, S_BUF, R_BUF)
#4 http_status <= #3.out 1
#5 header_start <= #3.out 2
#6 header_stop <= #3.out 3
#7 body_start <= #3.out 4
#8 body_stop <= #3.out 5
#9 http_get_done <= #3.out 6
#10 http_get_error <= #3.out 7
#11 DWORD_OF_BYTE(192, 168, 178, 001)
#12 IP_CONTROL_1:IP_CONTROL(#11, -, T#4s, IP_C, S_BUF, R_BUF)
#13 TON_1:TON(IN: http_get_done, PT: T#1s)
#14 http_release <= #13.Q
#15 COUNT_DR:COUNT_DR(-, -, http_get_done, -, -, -, -)
#16 cycles <= #15
#17 F_TRIG:F_TRIG(CLK: http_get_done)
#18 enable <= #17.Q
_END_CFC_
END_PROGRAM

(* POU INI_PARSER_BUF_DEMO, ST *)
PROGRAM INI_PARSER_BUF_DEMO
VAR
	STATION_NAME : STRING;
	STATION_IP : STRING;
	SMTP_SERVER : STRING;
	SMTP_FROM :	STRING;

	IPB : INI_PARSER_BUF;
	FS : FILE_SERVER;
	FSD : FILE_SERVER_DATA;
	PT : NETWORK_BUFFER;
	section : INT;
	key : STRING(STRING_LENGTH);
	value : STRING(STRING_LENGTH);
	str : STRING(STRING_LENGTH);
	step : INT;
	result : BYTE;
	offset : UDINT;
	run : BYTE;
	done : BOOL;

	FB_LOG_MESSAGE : LOG_MSG;
END_VAR
(* Demo-Programm: INI-Datei mittels Enumeration auswerten *)

(* ----- den nachfolgenden Textblock als datei "config.ini" auf der sps ablegen ---
# Demo - Initialisierungsdatei

[Station]
NAME=Test_Station_1
IP=192.168.178.1

[SMTP]
SERVER=test.server.de
FROM=test1@gmx.net
---------------------------------------------------------------------------------*)

CASE step OF

00:	IF NOT done THEN
	 	(* File_Daten einrichten  *)
		FSD.FILENAME := 'd:\pxc\oscat\network\config.ini'; (* Dateiname *)
		FSD.MODE := 1; (* vorhandene Datei zum lesen öffnen *)
		FSD.OFFSET := 0; (* Start bei Dateianfang *)
		FSD.AUTO_CLOSE := T#0s; (* kein Auto-Close verwenden *)
		PT.SIZE := 65535; (* maximale länge einlesen *)
		step := 10;
	END_IF;

10:	IF FSD.MODE = 0 THEN (* Datei geöffnet ? *)
		OFFSET := 0; (* Start Offset vorgeben *)
		str := '';
		run := 3; (* key suchen *)
		step := 20;
	END_IF;

20:	IF run = 0 THEN
		(* ---------------------- Debug-Message ----------------------------*)
		IF LOG_CL.ENABLE THEN
			LOG_CL.NEW_MSG := 'IPBD: /key >~1< /value >~2< /offset ~3 /Run ~4 /Result ~5';
			LOG_CL.PRINTF[1] := key;
			LOG_CL.PRINTF[2] := value;
			LOG_CL.PRINTF[3] := UDINT_TO_STRING(OFFSET);
			LOG_CL.PRINTF[4] := BYTE_TO_STRING(run);
			LOG_CL.PRINTF[5] := BYTE_TO_STRING(result);
			FB_LOG_MESSAGE();
		END_IF;
		(* -----------------------------------------------------------------*)

		run := 3; (* vorbelegung -> naechsten key suchen *)

		IF result = 1 THEN (* neue Sektion gefunden *)
			IF key = 'Station' THEN
				section := 1;
			ELSIF key = 'SMTP' THEN
				section := 2;

			(* hier können weitere Section hinzugefügt werden *)

			ELSE
				section := 0; (* unbekannte sektion gefunden -> ignorieren *)
			END_IF;

		ELSIF result = 2 AND section > 0 THEN (* Key in einer bekannten sektion gefunden *)

			CASE section OF

			1:  (* Section: Station *)
				IF key = 'NAME' THEN
					STATION_NAME := value; (* Name *)
				ELSIF key = 'IP' THEN
					STATION_IP := value; (* IP-Adresse *)
				END_IF;

				(* hier können weitere Schlüsselsauswertungen hinzugefügt werden *)

			2:  (* Section: SMTP *)
				IF key = 'SERVER' THEN
					SMTP_SERVER := value; (* SMTP Server *)
				ELSIF key = 'FROM' THEN
					SMTP_FROM := value; (* SMTP Absender *)
				END_IF;

				(* hier können weitere Schlüsselsauswertungen hinzugefügt werden *)

			END_CASE;

		ELSIF result = 10 THEN (* nichts mehr gefunden *)
			run := 0; (* keine weitere INI Auswertung erwünscht *)
			FSD.MODE := 5; (* Datei schliessen *)
			step := 30;
		END_IF;
	END_IF;

30:	IF FSD.MODE = 0 THEN (* Datei geschlossen ? *)
		step := 0;
		done := TRUE;
	END_IF;

END_CASE;

IPB(STR:=str,RUN:=run,OFFSET:=OFFSET,KEY:=key,VALUE:=value,PT:=PT); (* INI PARAMETER BUF *)
result:=IPB.RESULT;

FS(FSD:=FSD,PT:=PT); (* FILE_SERVER *)
END_PROGRAM

(* POU INI_PARSER_BUF, ST *)
FUNCTION_BLOCK INI_PARSER_BUF
VAR_IN_OUT
	STR : STRING(STRING_LENGTH);
	RUN : BYTE;
	OFFSET : UDINT;
	KEY : STRING(STRING_LENGTH);
	VALUE : STRING(STRING_LENGTH);
	PT : NETWORK_BUFFER;
END_VAR
VAR_OUTPUT
	RESULT : BYTE;
END_VAR
VAR
	step : INT;
	size : INT;
	c : BYTE;
	k_add : BYTE;
	v_add : BYTE;
	i : INT;
	state : BYTE;
	eof : BOOL;
	pv : POINTER TO BYTE;
	pk : POINTER TO BYTE;
	pve : DWORD;
	pke : DWORD;
	watchdog : TON;

	(*FB_LOG_MESSAGE : LOG_MSG;
	_debug_enable : BOOL := TRUE;
	step_last : INT;*)
END_VAR

(*
version 1.0		23. sep. 2010
programmer 		ks
tested by			ks

INI_PARSER_BUF liefert die Elemente einer Initialisierungsdatei die in einem Bytearray abgelegt ist.

--------------------------------------

RUN Mode
00 = kein Befehl aktiv
01 = Section melden
02 = Key melden
03 = Section oder Key melden

Result Codes
01 = Section gefunden
02 = Key gefunden
05 = Befehl in Arbeit (Busy)
10 = nichts gefunden - Daten-Ende erreicht
11 = keinen Key gefunden - Section-Ende erreicht

State Codes
00 = Indexüberschreitung - Bufferende
01 = Section gefunden
02 = Key gefunden
03 = Kommentar gefunden
05 = Befehl in Arbeit (Busy)
10 = nichts gefunden - Daten-Ende erreicht

*)
IF RUN > 0 THEN
	IF state = 0 THEN (* Auswertung neu beginnen *)

		pv := ADR(VALUE);
		pv^ := 0; (* VALUE = '' *)
		pve := pv + INT_TO_DWORD(STRING_LENGTH);
		pk := ADR(KEY);
		pk^ := 0; (* KEY = '' *)
		pke := pk + INT_TO_DWORD(STRING_LENGTH);

		i := UDINT_TO_INT(OFFSET);
		size := UINT_TO_INT(PT.SIZE) - 1;
		RESULT := 0;
		state := 5; (* Befehl in Arbeit (Busy) *)
		step := 0; (* Auswertung neu beginnen *)

		(* ---------------- Debug-Message -----------------------*)
		(*IF _debug_enable THEN
			LOG_CL.NEW_MSG := 'IPB: Startindex: ~1';
			LOG_CL.PRINTF[1]  := INT_TO_STRING(i);
			FB_LOG_MESSAGE();
		END_IF;*)
		(* -----------------------------------------------------------------*)
	END_IF;

	watchdog(IN:=FALSE,PT:=T#1ms); (* Timer neustarten *)
	watchdog.IN := TRUE;

	WHILE (state = 5) DO (* Schleife solange kein Ergebnis *)

		watchdog(); (* Timer aktualisieren *)

		IF watchdog.Q THEN (* watchdog ausgelöst *)
			state := 5;
			EXIT;
		ELSIF i > size THEN (* kein weiteres zeichen vorhanden *)
			state := 10; (* nichts gefunden - Daten-Ende erreicht *)
			EXIT;
		ELSE

			c := PT.BUFFER[i]; (* neues Zeichen aus Buffer lesen *)
			eof := i + 1 = PT.SIZE; (* End of File *)

			k_add := 0;
			v_add := 0;

			CASE step OF

			0: (* noch kein Modus erkannt *)
				IF c = 91 THEN (* mit "[" vergleichen *)
					step := 200; (* Modus für Section aktivieren *)
				ELSIF c = 59 OR c = 35 THEN (* mit ";" und '#' vergleichen *)
					step := 100; (* Modus für Kommentar aktivieren *)
				ELSIF c > 32 THEN (* Key erkannt *)
					k_add := c; (* Zeichen ablegen *)
					step := 300; (* Key auswertung starten *)
				END_IF;
			100: (* Kommentar erkannt -> Zeilenende suchen *)
				IF c < 32 THEN (* prüfe auf Steuerzeichen *)
					state  := 3; (* Beenden -> Kommentar wurde gefunden *)
				END_IF;
			200: (* Sections-start erkannt -> Sectionsende suchen *)
				IF c = 93 THEN (* mit "]" vergleichen *)
					IF pk > ADR(KEY) > 0 THEN (* innerhalb von [] muss sich mindestens ein Zeichen befinden *)
						state  := 1; (* Beenden -> Section wurde gefunden *)
					ELSE
						pk := ADR(KEY);
						pk^ := 0; (* KEY = '' *)
						step := 0; (* fehlerhafte Section-Zeile vorhanden -> weitersuchen *)
					END_IF;
				ELSIF c < 32 OR eof THEN (* Steuerzeichen - fehlerhafte Section-Zeile -> weitersuchen *)
					pk := ADR(KEY);
					pk^ := 0; (* KEY = '' *)
					step := 0;
				ELSE
					k_add := c; (* Zeichen ablegen *)
				END_IF;
			300: (* Beginn: Key erkannt -> Name auswerten *)
				IF c < 32 THEN (* Steuerzeichen - fehlerhafte Key-Zeile -> weitersuchen *)
					pk := ADR(KEY);
					pk^ := 0; (* KEY = '' *)
					step := 0;
				ELSIF c = 61 THEN (* prüfe auf '=' *)
					step := 330;
				ELSE
					k_add := c; (* Zeichen ablegen *)
				END_IF;
			330: (* KeyValue beginn suchen *)
				IF c < 32 THEN (* Steuerzeichen  *)
					state := 2; (* Key ohne Value gefunden *)
				ELSIF eof THEN
					state := 2; (* Key ohne Value gefunden *)
					v_add := c; (* Zeichen ablegen *)
				ELSE
					v_add := c; (* Zeichen ablegen *)
					step := 350;
				END_IF;
			350: (* KeyValue Ende suchen *)
				IF c < 32 THEN (* Steuerzeichen *)
					state := 2; (* Key gefunden *)
				ELSIF eof THEN
					v_add := c; (* Zeichen ablegen *)
					state := 2; (* Key gefunden *)
				ELSE
					v_add := c; (* Zeichen ablegen *)
				END_IF;
			END_CASE;

			IF v_add > 0  AND pv < pve THEN (* Zeichen zu Value-String hinzufügen *)
				pv^ := v_add; (* Zeichen eintragen *)
				pv := pv + 1;
				pv^ := 0; (* String-Terminierung eintragen *)
			END_IF;

			IF k_add > 0 AND pk < pke THEN (* Zeichen zu Key-String hinzufügen *)
				pk^ := k_add; (* Zeichen eintragen *)
				pk := pk + 1;
				pk^ := 0; (* String-Terminierung eintragen *)
			END_IF;

			i := i + 1; (* Datenzeiger erhöhen *)

		END_IF;
	END_WHILE;

	CASE state OF
	01:	(* Section gefunden *)
		IF RUN = 1 OR RUN = 3 THEN (* Section vorgewählt oder alles rückmelden *)
			IF KEY = STR OR LEN(STR) = 0 THEN (* mit gesuchter Section vergleichen oder keine Section vorgegeben *)
				RESULT := 1; (* Section gefunden *)
				OFFSET := i; (* Offset uebernehmen *)
				RUN := 0;
				state := 0;
			END_IF;
		ELSE
			pk := ADR(KEY);
			pk^ := 0; (* KEY = '' *)
			RESULT := 11; (* Key nicht gefunden , Section-Ende - Offset nicht verändern *)
			RUN := 0;
			state := 0;
		END_IF;
	02:	(* Key gefunden *)
		IF RUN = 2 OR RUN = 3 THEN (* Key vorgewählt oder alles rückmelden *)
			IF KEY = STR OR LEN(STR) = 0 THEN (* mit gesuchten Key vergleichen *)
				RESULT := 2; (* Key gefunden *)
				OFFSET := i; (* Offset uebernehmen *)
				RUN := 0;
				state := 0;
			END_IF;
		END_IF;
	03:	(* Kommenar gefunden *)
		OFFSET := i; (* Offset uebernehmen *)
		state := 0;

	05:	RESULT := 5; (* in Arbeit *)

	10:	(* Indexüberschreitung - Bufferende *)
		RESULT := 10; (* nichts gefunden - Datenende erreicht *)
		OFFSET := i; (* Offset uebernehmen *)
		RUN := 0;
		state := 0;
	END_CASE;

	(* ---------------- Debug-Message -----------------------*)
	(*IF _debug_enable THEN
		LOG_CL.NEW_MSG := 'IPF: intern Result ~1 , state ~2, step ~3 , offset ~4, run ~5';
		LOG_CL.PRINTF[1] := BYTE_TO_STRING(RESULT);
		LOG_CL.PRINTF[2] := BYTE_TO_STRING(state);
		LOG_CL.PRINTF[3] := INT_TO_STRING(step);
		LOG_CL.PRINTF[4] := UDINT_TO_STRING(OFFSET);
		LOG_CL.PRINTF[5] := BYTE_TO_STRING(RUN);
		FB_LOG_MESSAGE();
	END_IF;*)
	(* -----------------------------------------------------------------*)

END_IF;

(* ---------------- Debug-Message -----------------------*)
(*IF _debug_enable THEN
	IF step_last <> step THEN
		LOG_CL.NEW_MSG := 'IPB: Step: ~1';
		LOG_CL.PRINTF[1]  := INT_TO_STRING(step);
		FB_LOG_MESSAGE();
	END_IF;
	step_last := step;
END_IF;*)
(* -----------------------------------------------------------------*)

(* revision history
ks	23. sep. 2010	rev 1.0
	original version
*)
END_FUNCTION_BLOCK

(* POU INI_PARSER_FILE_DEMO, ST *)
PROGRAM INI_PARSER_FILE_DEMO
VAR
	STATION_NAME : STRING;
	STATION_IP : STRING;
	SMTP_SERVER : STRING;
	SMTP_FROM : STRING;

	IPF : INI_PARSER_FILE;
	FS : FILE_SERVER;
	FSD : FILE_SERVER_DATA;
	PT : NETWORK_BUFFER;
	section : INT;
	filename : STRING;
	key : STRING(STRING_LENGTH);
	value :	STRING(STRING_LENGTH);
	str : STRING(STRING_LENGTH);
	step : INT;
	result : BYTE;
	offset : UDINT;
	run : BYTE;
	done : BOOL;
	FB_LOG_MESSAGE : LOG_MSG;
END_VAR
(* Demo-Programm: INI-Datei mittels Enumeration auswerten *)

(* ----- den nachfolgenden Textblock als datei "config.ini" auf der sps ablegen ---
# Demo - Initialisierungsdatei

[Station]
NAME=Test_Station_1
IP=192.168.178.1

[SMTP]
SERVER=test.server.de
FROM=test1@gmx.net
---------------------------------------------------------------------------------*)

CASE step OF

00:	IF NOT done THEN
		filename := 'd:\pxc\oscat\network\config.ini'; (* File_Daten einrichten *)
		OFFSET := 0; (* Start Offset vorgeben *)
		FSD.AUTO_CLOSE := T#0ms; (* kein Automatisches schliessen *)
		str := '';
		run := 3; (* key suchen *)
		step := 20;
	END_IF;

20:	IF run = 0 THEN (* kein Befehl mehr aktiv ? *)
		(* ---------------------- Debug-Message ----------------------------*)
		IF LOG_CL.ENABLE THEN
			LOG_CL.NEW_MSG := 'IPFD: /key >~1< /value >~2< /offset ~3 /Run ~4 /Result ~5';
			LOG_CL.PRINTF[1] := key;
			LOG_CL.PRINTF[2] := value;
			LOG_CL.PRINTF[3] := UDINT_TO_STRING(OFFSET);
			LOG_CL.PRINTF[4] := BYTE_TO_STRING(run);
			LOG_CL.PRINTF[5] := BYTE_TO_STRING(result);
			FB_LOG_MESSAGE();
		END_IF;
		(* -----------------------------------------------------------------*)

		run := 3; (* vorbelegung -> naechsten key suchen *)

		IF result = 1 THEN (* neue Sektion gefunden *)
			IF key = 'Station' THEN
				section := 1;
			ELSIF key = 'SMTP' THEN
				section := 2;

			(* hier können weitere Section hinzugefügt werden *)

			ELSE
				section := 0; (* unbekannte sektion gefunden -> ignorieren *)
			END_IF;

		ELSIF result = 2 AND section > 0 THEN (* Key in einer bekannten sektion gefunden *)

			CASE section OF

			1:  (* Section: Station *)
				IF key = 'NAME' THEN
					STATION_NAME := value; (* Name *)
				ELSIF key = 'IP' THEN
					STATION_IP := value; (* IP-Adresse *)
				END_IF;

				(* hier können weitere Schlüsselsauswertungen hinzugefügt werden *)

			2:  (* Section: SMTP *)
				IF key = 'SERVER' THEN
					SMTP_SERVER := value; (* SMTP Server *)
				ELSIF key = 'FROM' THEN
					SMTP_FROM := value; (* SMTP Absender *)
				END_IF;

				(* hier können weitere Schlüsselsauswertungen hinzugefügt werden *)

			END_CASE;

		ELSIF result = 10 THEN (* nichts mehr gefunden *)
			run := 0; (* keine weitere INI Auswertung erwünscht *)
			FSD.MODE := 5; (* Datei schliessen *)
			step := 30;
		END_IF;
	END_IF;

30:	IF FSD.MODE = 0 THEN (* Befehl Datei schliessen beendet *)
		step := 0;
		done := TRUE;
	END_IF;

END_CASE;

IPF(FILENAME:=FILENAME,FSD:=FSD,STR:=str,RUN:=run,OFFSET:=OFFSET,KEY:=key,VALUE:=value,PT:=PT); (* INI PARAMETER FILE *)
result:=IPF.RESULT;

FS(FSD:=FSD,PT:=PT); (* FILE_SERVER *)
END_PROGRAM

(* POU INI_PARSER_FILE, ST *)
FUNCTION_BLOCK INI_PARSER_FILE
VAR_IN_OUT
	FILENAME : STRING;
	FSD : FILE_SERVER_DATA	;
	STR : STRING(STRING_LENGTH);
	RUN : BYTE;
	OFFSET : UDINT;
	KEY : STRING(STRING_LENGTH);
	VALUE : STRING(STRING_LENGTH);
	PT	: NETWORK_BUFFER;
END_VAR
VAR_OUTPUT
	RESULT : BYTE;
END_VAR
VAR
	FB : FILE_BLOCK;
	i : UDINT;
	state : BYTE;
	e : BYTE;
	mode : BYTE;
	step : INT;
	c : BYTE;
	k_add : BYTE;
	v_add : BYTE;
	eof : BOOL;
	pv : POINTER TO BYTE;
	pk : POINTER TO BYTE;
	pve : DWORD;
	pke : DWORD;
	watchdog : TON;

	(*FB_LOG_MESSAGE : LOG_MSG;
	_debug_enable : BOOL := TRUE;
	step_last : INT;*)
END_VAR

(*
version 1.0		23. sep. 2010
programmer 		ks
tested by			ks

INI_PARSER_FILE liefert die Elemente einer Initialisierungsdatei.

--------------------------------------

RUN Mode
00 = kein Befehl aktiv
01 = Section melden
02 = Key melden
03 = Section oder Key melden

Result Codes
01 = Section gefunden
02 = Key gefunden
05 = Befehl in Arbeit (Busy)
10 = nichts gefunden - Daten-Ende erreicht
11 = keinen Key gefunden - Section-Ende erreicht

State Codes
00 = Indexüberschreitung - Bufferende
01 = Section gefunden
02 = Key gefunden
03 = Kommentar gefunden
05 = Befehl in Arbeit (Busy)
10 = nichts gefunden - Daten-Ende erreicht

*)
IF RUN > 0 THEN

	IF state = 0 THEN (* Auswertung neu beginnen *)
		pv := ADR(VALUE);
		pv^ := 0; (* VALUE = '' *)
		pve := pv + INT_TO_DWORD(STRING_LENGTH);
		pk := ADR(KEY);
		pk^ := 0; (* KEY = '' *)
		pke := pk + INT_TO_DWORD(STRING_LENGTH);

		i := OFFSET;
		RESULT := 0;
		state := 5; (* Befehl in Arbeit (Busy) *)
		step := 0; (* Auswertung neu beginnen *)

		(* ---------------- Debug-Message -----------------------*)
		(*IF _debug_enable THEN
			LOG_CL.NEW_MSG := 'IPF: Startindex: ~1';
			LOG_CL.PRINTF[1] := UDINT_TO_STRING(i);
			FB_LOG_MESSAGE();
		END_IF;*)
		(* -----------------------------------------------------------------*)

	END_IF;

	watchdog(IN:=FALSE,PT:=T#1ms); (* Timer neustarten *)
	watchdog.IN := TRUE;

	WHILE (state = 5) DO (* Schleife solange kein Ergebnis *)

		mode := 1;
		FB(MODE:=mode,FSD:=fsd,PT:=PT,FILENAME:=FILENAME,POS:=i );
		e:=FB.ERROR;
		c:=FB.DATA;

		eof := i + 1 = FSD.FILE_SIZE; (* End of File *)

		(* ---------------- Debug-Message -----------------------*)
		(*IF _debug_enable THEN
			LOG_CL.NEW_MSG := 'IPF: mode: ~1, error: ~2 , >~7<>~3< ~4 step ~5 index ~6';
			LOG_CL.PRINTF[1] := BYTE_TO_STRING(mode);
			LOG_CL.PRINTF[2] := BYTE_TO_STRING(e);
			LOG_CL.PRINTF[3] := BYTE_TO_STRING(c);
			LOG_CL.PRINTF[4] := BOOL_TO_STRING(eof);
			LOG_CL.PRINTF[5] := INT_TO_STRING(step);
			LOG_CL.PRINTF[6] := UDINT_TO_STRING(i);
			LOG_CL.PRINTF[7] := CHR_TO_STRING(c);
			FB_LOG_MESSAGE();
		END_IF;*)
		(* -----------------------------------------------------------------*)
		watchdog(); (* Timer aktualisieren *)

		IF mode > 0 OR watchdog.Q THEN (* Baustein noch aktiv, oder watchdog ausgelöst *)
			state := 5;
			EXIT;
		ELSIF e > 0 THEN (* File_error oder kein weiteres zeichen vorhanden *)
			state := 10; (* nichts gefunden - Daten-Ende erreicht *)
			EXIT;
		ELSE

			k_add := 0;
			v_add := 0;

			CASE step OF

			0: (* noch kein Modus erkannt *)
				IF c = 91 THEN (* mit "[" vergleichen *)
					step := 200; (* Modus für Section aktivieren *)
				ELSIF c = 59 OR c = 35 THEN (* mit ";" und '#' vergleichen *)
					step := 100; (* Modus für Kommentar aktivieren *)
				ELSIF c > 32 THEN (* Key erkannt *)
					k_add := c; (* Zeichen ablegen *)
					step := 300; (* Key auswertung starten *)
				END_IF;
			100: (* Kommentar erkannt -> Zeilenende suchen *)
				IF c < 32 THEN (* prüfe auf Steuerzeichen *)
					state  := 3; (* Beenden -> Kommentar wurde gefunden *)
				END_IF;
			200: (* Sections-start erkannt -> Sectionsende suchen *)
				IF c = 93 THEN (* mit "]" vergleichen *)
					IF pk > ADR(KEY) > 0 THEN (* innerhalb von [] muss sich mindestens ein Zeichen befinden *)
						state  := 1; (* Beenden -> Section wurde gefunden *)
					ELSE
						pk := ADR(KEY);
						pk^ := 0; (* KEY = '' *)
						step := 0; (* fehlerhafte Section-Zeile vorhanden -> weitersuchen *)
					END_IF;
				ELSIF c < 32 OR eof THEN (* Steuerzeichen - fehlerhafte Section-Zeile -> weitersuchen *)
					pk := ADR(KEY);
					pk^ := 0; (* KEY = '' *)
					step := 0;
				ELSE
					k_add := c; (* Zeichen ablegen *)
				END_IF;
			300: (* Beginn: Key erkannt -> Name auswerten *)
				IF c < 32 THEN (* Steuerzeichen - fehlerhafte Key-Zeile -> weitersuchen *)
					pk := ADR(KEY);
					pk^ := 0; (* KEY = '' *)
					step := 0;
				ELSIF c = 61 THEN (* prüfe auf '=' *)
					step := 330;
				ELSE
					k_add := c; (* Zeichen ablegen *)
				END_IF;
			330: (* KeyValue beginn suchen *)
				IF c < 32 THEN (* Steuerzeichen  *)
					state := 2; (* Key ohne Value gefunden *)
				ELSIF eof THEN
					state := 2; (* Key ohne Value gefunden *)
					v_add := c; (* Zeichen ablegen *)
				ELSE
					v_add := c; (* Zeichen ablegen *)
					step := 350;
				END_IF;
			350: (* KeyValue Ende suchen *)
				IF c < 32 THEN (* Steuerzeichen *)
					state := 2; (* Key gefunden *)
				ELSIF eof THEN
					v_add := c; (* Zeichen ablegen *)
					state := 2; (* Key gefunden *)
				ELSE
					v_add := c; (* Zeichen ablegen *)
				END_IF;
			END_CASE;

			IF v_add > 0  AND pv < pve THEN (* Zeichen zu Value-String hinzufügen *)
				pv^ := v_add; (* Zeichen eintragen *)
				pv := pv + 1;
				pv^ := 0; (* String-Terminierung eintragen *)
			END_IF;

			IF k_add > 0 AND pk < pke THEN (* Zeichen zu Key-String hinzufügen *)
				pk^ := k_add; (* Zeichen eintragen *)
				pk := pk + 1;
				pk^ := 0; (* String-Terminierung eintragen *)
			END_IF;

			i := i + 1; (* Datenzeiger erhöhen *)

		END_IF;
	END_WHILE;

	CASE state OF
	01:	(* Section gefunden *)
		IF RUN = 1 OR RUN = 3 THEN (* Section vorgewählt oder alles rückmelden *)
			IF KEY = STR OR LEN(STR) = 0 THEN (* mit gesuchter Section vergleichen oder keine Section vorgegeben *)
				RESULT := 1; (* Section gefunden *)
				OFFSET := i; (* Offset uebernehmen *)
				RUN := 0;
				state := 0;
			END_IF;
		ELSE
			pk := ADR(KEY);
			pk^ := 0; (* KEY = '' *)
			RESULT := 11; (* Key nicht gefunden , Section-Ende - Offset nicht verändern *)
			RUN := 0;
			state := 0;
		END_IF;
	02:	(* Key gefunden *)
		IF RUN = 2 OR RUN = 3 THEN (* Key vorgewählt oder alles rückmelden *)
			IF KEY = STR OR LEN(STR) = 0 THEN (* mit gesuchten Key vergleichen *)
				RESULT := 2; (* Key gefunden *)
				OFFSET := i; (* Offset uebernehmen *)
				RUN := 0;
				state := 0;
			END_IF;
		END_IF;
	03:	(* Kommenar gefunden *)
		OFFSET := i; (* Offset uebernehmen *)
		state := 0;

	05:	RESULT := 5; (* in Arbeit *)

	10:	(* Indexüberschreitung - Bufferende *)
		RESULT := 10; (* nichts gefunden - Datenende erreicht *)
		OFFSET := i; (* Offset uebernehmen *)
		RUN := 0;
		state := 0;
	END_CASE;

	(* ---------------- Debug-Message -----------------------*)
	(*IF _debug_enable THEN
		LOG_CL.NEW_MSG := 'IPF: intern Result ~1 , state ~2, step ~3 , offset ~4, run ~5';
		LOG_CL.PRINTF[1] := BYTE_TO_STRING(RESULT);
		LOG_CL.PRINTF[2] := BYTE_TO_STRING(state);
		LOG_CL.PRINTF[3] := INT_TO_STRING(step);
		LOG_CL.PRINTF[4] := UDINT_TO_STRING(OFFSET);
		LOG_CL.PRINTF[5] := BYTE_TO_STRING(RUN);
		FB_LOG_MESSAGE();
	END_IF;*)
	(* -----------------------------------------------------------------*)

END_IF;

(* ---------------- Debug-Message -----------------------*)
(*IF _debug_enable THEN
	IF step_last <> step THEN
		LOG_CL.NEW_MSG := 'IPB: Step: ~1';
		LOG_CL.PRINTF[1]  := INT_TO_STRING(step);
		FB_LOG_MESSAGE();
	END_IF;
	step_last := step;
END_IF;*)
(* -----------------------------------------------------------------*)

(* revision history
ks	23. sep. 2010	rev 1.0
	original version
*)
END_FUNCTION_BLOCK

(* POU IP2GEO_DEMO, CFC *)
PROGRAM IP2GEO_DEMO
VAR
	IP_C: IP_C;
	S_BUF: NETWORK_BUFFER;
	R_BUF: NETWORK_BUFFER;
	IP_CONTROL_1: IP_CONTROL;
	TON_1: TON;
	IP2GEO_1: IP2GEO;
	COUNT_DR_1: COUNT_DR;
	GEO: IP2GEO_DATA;
	activate: BOOL := TRUE;
	done: BOOL;
	count_cycles: DWORD;
	busy: BOOL;
	error_c: DWORD;
	error_t: BYTE;
	cwtime: TIME;
END_VAR
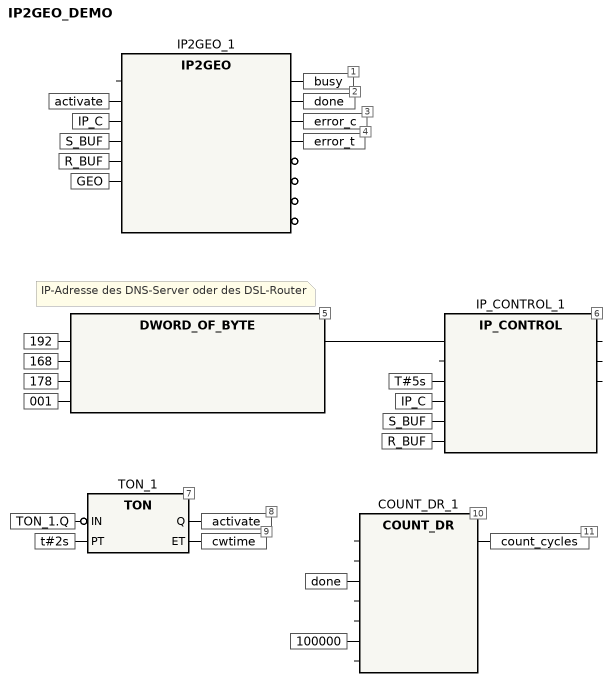
_CFC_ (* Continuous Function Chart, elements in execution order *)
(* IP-Adresse des DNS-Server oder des DSL-Router *)
#0 IP2GEO_1:IP2GEO(-, activate, IP_C, S_BUF, R_BUF, GEO)
#1 busy <= #0.out 1
#2 done <= #0.out 2
#3 error_c <= #0.out 3
#4 error_t <= #0.out 4
#5 DWORD_OF_BYTE(192, 168, 178, 001)
#6 IP_CONTROL_1:IP_CONTROL(#5, -, T#5s, IP_C, S_BUF, R_BUF)
#7 TON_1:TON(IN: NOT TON_1.Q, PT: t#2s)
#8 activate <= #7.Q
#9 cwtime <= #7.ET
#10 COUNT_DR_1:COUNT_DR(-, -, done, -, -, 100000, -)
#11 count_cycles <= #10
_END_CFC_
END_PROGRAM

(* POU IP2GEO, ST *)
FUNCTION_BLOCK IP2GEO
VAR_IN_OUT
	IP_C : IP_C; (* IP_Control Verwaltungsstruktur *)
	S_BUF : NETWORK_BUFFER;
	R_BUF : NETWORK_BUFFER;
	GEO : IP2GEO_DATA;
END_VAR
VAR_INPUT
	IP : DWORD;
	ACTIVATE : BOOL;
END_VAR
VAR_OUTPUT
	BUSY : BOOL;
	DONE : BOOL;
	ERROR_C : DWORD;
	ERROR_T : BYTE;
END_VAR
VAR
	CTRL : XML_CONTROL;
	XML_READER : XML_READER;
	URL_DATA : url;
	DNS_CLIENT : DNS_CLIENT;
	HTTP_GET : HTTP_GET;
	last_state : BOOL;
	value_int :	INT;
	value_real : REAL;
	v_real : REAL;
	state : INT;
END_VAR
(*

version 	1.1	07.oct. 2010
programmer 	ks
tested by	ks

IP2GEO ermittelt die aktuelle WAN-IP und die dazugehörigen geographischen Infos

zusatzinfos: http://www.worldtimezone.com/time/wtzresult.php?CiID=10182&forma=

example:

http://ipinfodb.com/ip_query.php?timezone=true&IP=

<?xml version="1.0" encoding="UTF-8" ?> 
- <Response>
  <Ip>85.127.218.109</Ip> 
  <Status>OK</Status> 
  <CountryCode>AT</CountryCode> 
  <CountryName>Austria</CountryName> 
  <RegionCode>09</RegionCode> 
  <RegionName>Wien</RegionName> 
  <City>Vienna</City> 
  <ZipPostalCode /> 
  <Latitude>48.2</Latitude> 
  <Longitude>16.3667</Longitude> 
  <TimezoneName>Europe/Vienna</TimezoneName> 
  <Gmtoffset>7200</Gmtoffset> 
  <Isdst>1</Isdst> 
  </Response>

*)
CASE state OF

00:
	IF ACTIVATE AND NOT last_state THEN
		state := 20;
		DONE := FALSE;
		BUSY := TRUE;
		ERROR_C := DWORD#0;
		ERROR_T := BYTE#0;
	END_IF;

20: (* URL for DNS UND HTTP-GET *)
	(* Example: http://ipinfodb.com/ip_query.php?ip=10.10.10.10 *)
	(* Example: http://ipinfodb.com/ip_query.php?timezone=true&IP=*)
	URL_DATA:=STRING_TO_URL(STR:='http://ipinfodb.com/ip_query.php?timezone=true&IP=',DEFAULT_PROTOCOL:='',DEFAULT_PATH:='');

	IF IP > DWORD#0 THEN
		URL_DATA.QUERY := CONCAT(URL_DATA.QUERY,IP4_TO_STRING(IP4:=IP));
	END_IF;

	state := 40;

40:
	IF DNS_CLIENT.DONE THEN
		state := 60;
	ELSIF (DNS_CLIENT.ERROR > DWORD#00) THEN
		(* Fehlerbehandlung *)
		ERROR_C := DNS_CLIENT.ERROR;
		ERROR_T := BYTE#01;
		state := 100;
	END_IF;

60:
	IF HTTP_GET.DONE THEN
		state := 80;
		CTRL.START_POS := HTTP_GET.BODY_START;
		CTRL.STOP_POS := HTTP_GET.BODY_STOP;
		CTRL.COMMAND := WORD#2#10000000_00011000; (* ONLY TEXT AND ATTRIBUTE *)
		CTRL.WATCHDOG := T#1ms;

	ELSIF (HTTP_GET.ERROR > DWORD#00) THEN
		(* Fehlerbehandlung *)
		ERROR_C := HTTP_GET.ERROR;
		ERROR_T := BYTE#02;
		state := 100;
	END_IF;

80:
	(* XML Daten seriell lesen *)
	XML_READER(CTRL:=CTRL,BUF:=R_BUF.BUFFER);
	IF CTRL.TYP < 98 THEN (* nur auswerten wenn kein Watchdog durchlauf *)
		(* automatische konvertierung in real und int ausführen *)
		value_int := 0;
		value_real := 0.0;
		IF LEN(CTRL.VALUE) <= 20 THEN
			v_real :=FLOAT_TO_REAL(FLT:=CTRL.VALUE);
			IF CHK_REAL(v_real) = 0 THEN (* !!! prüft auf gültigen REAL Wert, ansonsten stürzt Twincat ab !!!!  *)
				value_real := v_real;
				value_int := REAL_TO_INT(value_real);
			END_IF;
		END_IF;

		CASE UINT_TO_INT(CTRL.COUNT) OF

		07: GEO.IP4 := IP4_DECODE(STR:=CTRL.VALUE); (* IP-Adresse *)
		10: GEO.STATE := 'OK' = CTRL.VALUE; (* STATUS *)
		13: GEO.COUNTRY_CODE := CTRL.VALUE; (* Country-Code *)
		16: GEO.COUNTRY_NAME := CTRL.VALUE; (* Country-Name *)
		19: GEO.REGION_CODE := CTRL.VALUE; (* Region-Code *)
		22: GEO.REGION_NAME := CTRL.VALUE; (* Region-Name *)
		25: GEO.CITY := CTRL.VALUE; (* City *)
		31: GEO.GEO_LATITUDE := value_real; (* Latitude *)
		34: GEO.GEO_LONGITUDE := value_real; (* Longitude *)
		37: GEO.TIME_ZONE_NAME := CTRL.VALUE; (* TimeZone Name *)
		40: GEO.GMT_OFFSET := value_int; (* GMT OFFSET in Sekunden *)
		43: GEO.IS_DST := value_int > 0; (* Sommerzeit aktiv *)
		END_CASE;

	ELSIF CTRL.TYP = 99 THEN (* EXIT - letztes Element gelesen *)
		DONE := TRUE;
		state := 100;
	END_IF;

100:
	(* UNLOCK HTTP DATA *)
	IF (NOT HTTP_GET.DONE) THEN
		state := 0;
		BUSY := FALSE;
		DONE := ERROR_T = BYTE#0;
	END_IF;

END_CASE;

(* ---------------- DNS --------------- *)
DNS_CLIENT(	IP_C:=IP_C,
			S_BUF:=S_BUF,
			R_BUF:=R_BUF,
			DOMAIN:=URL_DATA.DOMAIN,
			IP4_DNS:=DWORD#00,
			ACTIVATE:=state=40 (* DNS Start *)
			);

(* nicht oder nicht direkt verwendete Parameter *)
(* 	DWORD :=DNS_CLIENT.IP4;
	BOOL  :=DNS_CLIENT.DONE;
	BYTE  :=DNS_CLIENT.ERROR; *)
(* -------------------------------------*)

(* ------------- HTTP_GET --------------- *)
HTTP_GET(	IP_C:=IP_C,
			S_BUF:=S_BUF,
			R_BUF:=R_BUF,
			IP4:=DNS_CLIENT.IP4,
			GET:=state=60,
			MODE:=BYTE#2, (* HTTP 1.1 mit persistenter Verbindung *)
			UNLOCK_BUF:=state=100,
			URL_DATA:=URL_DATA
			);

(* nicht oder nicht direkt verwendete Parameter *)
(*	STRING := HTTP_GET.HTTP_STATUS;
	UINT :=HTTP_GET.HEADER_START;
	UINT :=HTTP_GET.HEADER_STOP;
	UINT :=HTTP_GET.BODY_START;
	UINT :=HTTP_GET.BODY_STOP;
	BOOL :=HTTP_GET.DONE;
	BYTE :=HTTP_GET.ERROR;
*)
(* -------------------------------------*)

last_state := ACTIVATE;

(* revision history
ks	14. aug. 2009	rev 1.0
	original version

ks	07. oct. 2010	rev 1.1
	new url , ip2geo fields , REAL_CHECK
*)
END_FUNCTION_BLOCK

(* POU XML_READER, ST *)
FUNCTION_BLOCK XML_READER
VAR_IN_OUT
	CTRL : XML_CONTROL;
	BUF : NW_BUF_LONG;
END_VAR
VAR
	index :	INT;
	index2 : INT;
	stop : INT;
	mode : INT;
	command : WORD;
	c :	BYTE;
	s1 : INT;
	e1 : INT;
	path_overflow : BOOL;
	empty_tag : BOOL;
	s_code : STRING(10);
	e_code : STRING(10);
	watchdog : TON;
END_VAR

(*

version 1.2		10. mai 2010
programmer 	ks
tested by		ks

XML_READER ermöglicht das serielle Parsen und die Auswertung von XML_Elementen in einem Buffer
*)
(*

TYP
00 = UNBEKANNT
01 = ELEMENT (STANDARD)
02 = CLOSE ELEMENT 
03 = TEXT
04 = ATTRIBUTE
05 = ELEMENT (PROCESSING INSTRUCTION) 

12 = !CDATA
13 = !COMMENT
14 = !DTD ELEMENT (Document Type Declarations )

98 = WATCHDOG
99 = ENDE

Bei Typ 02 werden keine Blockdaten ausgegeben !

*)

(* ---------- Init -------------- *)
IF BIT_OF_DWORD(WORD_TO_DWORD(CTRL.COMMAND),15) THEN
	COMMAND := CTRL.COMMAND;
	CTRL.COMMAND := WORD#0;

	index := UINT_TO_INT(CTRL.START_POS);
	stop := UINT_TO_INT(CTRL.STOP_POS);
	mode := 100;
	path_overflow := FALSE;

	CTRL.TYP := 0;
	CTRL.COUNT := UINT#00;
	CTRL.LEVEL := UINT#00;
	CTRL.ATTRIBUTE := '';
	CTRL.ELEMENT := '';
	CTRL.PATH := '';
	CTRL.VALUE := '';

	WATCHDOG.PT := CTRL.WATCHDOG;
END_IF;

(*----------------------------------------------- *)

IF index < 0 THEN RETURN;END_IF;

CTRL.BLOCK1_START := UINT#0;
CTRL.BLOCK1_STOP := UINT#0;
CTRL.BLOCK2_START := UINT#0;
CTRL.BLOCK2_STOP := UINT#0;

WATCHDOG(IN:=FALSE); (* Timer stoppen *)

WHILE (TRUE) DO

	(* -------------- WATCHDOG ------------------ *)
	WATCHDOG(IN:=CTRL.WATCHDOG > T#0s);
	IF WATCHDOG.Q THEN
		CTRL.TYP := 98;
		RETURN;
	END_IF;

	(* -------------- PARSING END ------------------ *)
	IF index > stop THEN
		CTRL.COUNT := CTRL.COUNT + UINT#1;
		CTRL.TYP := 99;
		mode  := 0; (* Schritt ruecksetzen *)
		index := 0; (* Abarbeitung stoppen *)
		RETURN;
	END_IF;

	CASE mode OF

	100: (* ---------- ELEMENT SECTION ------------------ *)
		(* search begin of element *)
		s1 := 0;
		e1 := 0;
		WHILE (index <= stop) DO
			IF BUF[INDEX]=BYTE#60 THEN (* '<' TagBegin *)
				index := index + 1;
				C := BUF[index];
				IF C = BYTE#47 THEN (* '/' TagTerm *)
					mode := 300; (* End Element Section *)
				ELSIF C = BYTE#33 THEN (* '!' for Special Section *)
					index := index + 1;
					mode := 500;
				ELSE
					s1 := index;
				END_IF;
				EXIT;
			END_IF;
			index := index + 1;
		END_WHILE;

		(* analyse element *)
		CTRL.TYP := 0; (* TYP löschen *)
		IF s1 > 0 THEN
			WHILE (index <= stop AND e1 = 0) DO
				c := BUF[index];
				(* whitespace zeichen = Element with Attributes *)
				IF c <= BYTE#32 THEN
					(* suche nächstes druckbares zeichen *)
					index2 := index;
					WHILE (index2 <= stop) AND (BUF[index2] <= BYTE#32) DO
						index2 := index2 + 1;
					END_WHILE;
					IF BUF[index2] = BYTE#47 THEN (* pruefe auf leeres Element '/' *)
						index := index2;
						e1 := index - 2;
						CTRL.TYP := 1; (* struktur-element *)
						mode := 300;   (* Close Element *)
						EXIT;
					END_IF;

					e1 := index - 1;
					CTRL.TYP := 1; (* Element mit Attribute *)
					mode := 400;

				ELSIF c = BYTE#62 THEN (* '>' TagEnd *)

					(* pruefe auf leeres Element <xx/> *)
					index2 := index - 1;
					IF BUF[index2] = BYTE#47 THEN (* TagTerm '/' *)
						e1 := index2 - 1;
						CTRL.TYP := 1;
						EMPTY_TAG := TRUE; (* EMPTY TAG Mode *)
						mode := 200; (* TEXT Element *)
						EXIT;
					END_IF;

					e1 := index - 1;
					index2 := index + 1;

					(* untersuche nachfolgendes Element *)
					WHILE (index2 <= stop) DO
						c := BUF[index2];
						IF c = BYTE#60 THEN (* '<' TagBegin *)

							index2 := index2 + 1; (* geht bei PCWORX leider nicht anders !*)
							c := BUF[index2];
							index2 := index2 - 1;
							IF c = BYTE#47 THEN (* TagTerm '/' *)
								empty_tag := TRUE;
								mode := 200; (* TEXT Element *)
							ELSE
								mode := 100; (* Element *)
							END_IF;
							CTRL.TYP := 1; (* struktur-element *)
							EXIT;
						ELSIF c > BYTE#32  THEN (* Printable-Character *)
							CTRL.TYP := 1; (* element with text *)
							mode := 200;
							EXIT;
						END_IF;
						index2 := index2 + 1;
					END_WHILE;
				END_IF;
				index := index + 1;
			END_WHILE;
		END_IF;

		(* Neues Element gefunden*)
		IF CTRL.TYP > 0 THEN

			(* Sonderprüfung auf Processing Instruction (PI) *)
			IF BUF[s1] = BYTE#63 THEN (* '?' for Processing Instruction *)
				s1 := s1 + 1; (* führendes '?' auslassen *)
				CTRL.TYP := 5;
			END_IF;
			CTRL.BLOCK1_START := INT_TO_UINT(s1);
			CTRL.BLOCK1_STOP  := INT_TO_UINT(e1);
			CTRL.ELEMENT := BUFFER_TO_STRING(PT:=ADR(BUF),SIZE:=INT_TO_UINT(stop + 1),START:=CTRL.BLOCK1_START,STOP:=CTRL.BLOCK1_STOP);
			CTRL.COUNT := CTRL.COUNT + UINT#1;
			CTRL.LEVEL := CTRL.LEVEL + UINT#1;

			IF path_overflow = FALSE THEN
				(* Stringlänge überwachen *)
				IF LEN(CTRL.PATH) + LEN(CTRL.ELEMENT) + 1 > 250 THEN
					path_overflow := TRUE;
					CTRL.PATH := 'OVERFLOW';
				ELSE
					CTRL.PATH := CONCAT(CTRL.PATH,'/');
					CTRL.PATH  := CONCAT(CTRL.PATH,CTRL.ELEMENT);
				END_IF;
			END_IF;

			IF BIT_OF_DWORD(WORD_TO_DWORD(COMMAND),CTRL.TYP) THEN
				RETURN;
			END_IF;
		END_IF;

	200: (* ---------- TEXT SECTION ------------------ *)
		CTRL.VALUE := '';
		IF empty_tag = FALSE THEN
			s1 := index;
			(* suche '<' EndTag*)
			WHILE (index <= stop) AND (BUF[index] <> BYTE#60) DO
				index := index + 1;
			END_WHILE;

			E1 := index - 1;
			CTRL.BLOCK1_START := INT_TO_UINT(s1);
			CTRL.BLOCK1_STOP  := INT_TO_UINT(e1);
			CTRL.VALUE := BUFFER_TO_STRING(PT:=ADR(BUF),SIZE:=INT_TO_UINT(stop + 1),START:=CTRL.BLOCK1_START,STOP:=CTRL.BLOCK1_STOP);
		END_IF;

		empty_tag := FALSE;
		mode := 300; (* -> NEXT-JOB: END ELEMENT *)
		CTRL.COUNT := CTRL.COUNT + UINT#1;
		CTRL.TYP := 3;

		IF BIT_OF_DWORD(WORD_TO_DWORD(command),CTRL.TYP) THEN
			RETURN;
		END_IF;

	300: (* ---------- END ELEMENT SECTION ------------------ *)
		WHILE (index <= stop) DO
			c := BUF[index];
			IF c = BYTE#62 THEN (* '>' TagEnd *)
				index := index + 1;
				s1 := FINDB(str1:=CTRL.PATH,str2:='/');
				IF path_overflow = FALSE THEN
					IF s1 > 1 THEN
						CTRL.ELEMENT := RIGHT(CTRL.PATH,LEN(CTRL.PATH) - s1);
						CTRL.PATH := LEFT(CTRL.PATH,s1 - 1);
					ELSE
						CTRL.ELEMENT := RIGHT(CTRL.PATH,LEN(CTRL.PATH) - 1);
						CTRL.PATH :='';
					END_IF;
				END_IF;

				CTRL.LEVEL := CTRL.LEVEL - UINT#1;
				CTRL.COUNT := CTRL.COUNT + UINT#1;
				CTRL.TYP := 2;
				mode := 100;

				IF BIT_OF_DWORD(WORD_TO_DWORD(COMMAND),CTRL.TYP) THEN
					RETURN;
				ELSE
					EXIT;
				END_IF;
			END_IF;
			index := index + 1;
		END_WHILE;

	400: (* ---------- ATTRIBUTE SECTION ------------------ *)
		(* search first normal charakter *)
		WHILE (index <= stop AND BUF[index] <= BYTE#32) DO
			index := index + 1;
		END_WHILE;

		(* begin Attribe name *)
		e1 := 0;
		s1 := index;
		(* search end of Attrib Name '=' *)
		WHILE (index <= stop) DO
			IF BUF[index] = BYTE#61 THEN (* '=' Equals *)
				e1 := index - 1;
				EXIT;
			END_IF;
			index := index + 1;
		END_WHILE;

		IF e1 > 0 THEN
			(* Attribute Name *)
			CTRL.BLOCK1_START := INT_TO_UINT(s1);
			CTRL.BLOCK1_STOP  := INT_TO_UINT(e1);
			CTRL.ATTRIBUTE := BUFFER_TO_STRING(PT:=ADR(BUF),SIZE:=INT_TO_UINT(STOP + 1),START:=CTRL.BLOCK1_START,STOP:=CTRL.BLOCK1_STOP);
			(* search end of Attrib Value '=' *)
			index := index + 2;
			e1 := 0;
			s1 := INDEX;
			WHILE (index <= stop AND e1 = 0) DO
				c := BUF[index];
				IF c = BYTE#34 OR c = BYTE#39 THEN (* " OR ' Equals *)
					e1 := index - 1;
				END_IF;
				index := index + 1;
			END_WHILE;

			IF e1 > 0 THEN
				(* Value *)
				CTRL.BLOCK2_START := INT_TO_UINT(s1);
				CTRL.BLOCK2_STOP  := INT_TO_UINT(e1);

				(* bei leeren "" ist start groesser als stop und wird somit zum leerstring *)
				CTRL.VALUE := BUFFER_TO_STRING(PT:=ADR(BUF),SIZE:=INT_TO_UINT(stop + 1),START:=CTRL.BLOCK2_START,STOP:=CTRL.BLOCK2_STOP);
				(* search next non white space charakter *)
				WHILE (index <= stop AND BUF[index] <= BYTE#32) DO
					index := index + 1;
				END_WHILE;

					c := BUF[index];
					(* TagEnd '>' *)
					IF c = BYTE#62 THEN
						index := index + 1;
						index2 := index;

					(* search next non white space charakter *)
					WHILE (index <= stop AND BUF[index] <= BYTE#32) DO
						index := index + 1;
					END_WHILE;

					IF BUF[index] = BYTE#60 THEN (* TagBegin '<' *)
						mode := 100; (* -> NEXT-JOB: ELEMENT-SECTION *)
					ELSE
						index := index2;
						mode := 200; (* -> NEXT-JOB: TEXT-SECTION *)
					END_IF;

				ELSIF c = BYTE#47 OR c = BYTE#63 THEN (* TagTerm '/' OR '?' end Processing Instruction *)
					mode := 300; (* -> NEXT-JOB: END ELEMENT *)
				ELSE
					mode := 400; (* -> NEXT-JOB: ATTRIBUTE-SECTION *)
				END_IF;

				CTRL.COUNT := CTRL.COUNT + UINT#1;
				CTRL.TYP := 4;
				IF BIT_OF_DWORD(WORD_TO_DWORD(command),CTRL.TYP) THEN
					RETURN;
				END_IF;
			END_IF;
		END_IF;

	500: (* ---------- SPECIAL DATA SECTION (Document Type Declarations) ---------- *)

		CTRL.TYP := 0;
		s1 := 0;
		index2 := 11;

		WHILE (s1 = 0) DO
			index2 := index2 + 1;
			CTRL.TYP := index2;

			CASE index2 OF
			12: (* CDATA *)
				s_code := '[CDATA[';
				e_code := ']]>';
			13: (* COMMENT *)
				s_code := '--';
				e_code := '-->';
			14: (* ANY DTD *)
				e_code := '';
				s1 := index;
				EXIT;
			END_CASE;

			e1 := LEN(s_code);
			IF BUFFER_SEARCH(PT:=ADR(BUF),SIZE:=INT_TO_UINT(index + e1),STR:=S_CODE,POS:=index,IGN:=FALSE) = INDEX THEN
				s1 := index + e1;
			END_IF;
		END_WHILE;

		CTRL.BLOCK1_START := INT_TO_UINT(s1);
		IF LEN(e_code) > 0 THEN
			(* Ende Kennung suchen *)
			e1 := BUFFER_SEARCH(PT:=ADR(BUF),SIZE:=INT_TO_UINT(stop + 1),STR:=e_code,POS:=index,IGN:=FALSE);
			CTRL.BLOCK1_STOP := INT_TO_UINT(e1 - 1);
			index := e1 + LEN(e_code); (* naechstes element *)
		ELSE
			(* suche '>' EndTag*)
			index2 := 1; (* <> Paar zähler *)
			WHILE (index <= stop AND index2 > 0) DO
				c := BUF[index];
				IF c = BYTE#60 THEN (* '<' TagBegin *)
					index2 := index2 + 1;
				ELSIF c = BYTE#62 THEN (* '>' TagEnd   *)
					index2 := index2 - 1;
				ELSIF c = BYTE#34 OR c = BYTE#39 THEN (* " Double Quote OR ' Single Quote *)
					index := index + 1;
					WHILE (index <= stop) DO
						c := BUF[index];
						IF c = BYTE#34 OR c = BYTE#39 THEN (* " Double Quote OR ' Single Quote *)
							EXIT;
						END_IF;
						index := index + 1;
					END_WHILE;
				END_IF;
				index := index + 1;
			END_WHILE;
			CTRL.BLOCK1_STOP := INT_TO_UINT(index - 2);
		END_IF;

		CTRL.VALUE := BUFFER_TO_STRING(PT:=ADR(BUF),SIZE:=INT_TO_UINT(stop + 1),START:=CTRL.BLOCK1_START,STOP:=CTRL.BLOCK1_STOP);
		CTRL.COUNT := CTRL.COUNT + UINT#1;
		mode := 100; (* -> NEXT-JOB: ELEMENT *)

		IF BIT_OF_DWORD(WORD_TO_DWORD(command),CTRL.TYP) THEN
			RETURN;
		END_IF;

	END_CASE;
END_WHILE;


(* revision history
ks	18. oct. 2008	rev 1.0
	original version

ks	20. oct. 2009	rev 1.1
	Networkbuffer und Buffer-funktionen auf Basis 0

ks	10. mai. 2010	rev 1.2
	stringlänge maximal 250 zeichen

*)
END_FUNCTION_BLOCK

(* POU IRTRANS_DEMO, CFC *)
PROGRAM IRTRANS_DEMO
VAR
	IP_C : IP_C;
	S_BUF : NETWORK_BUFFER_SHORT;
	R_BUF : NETWORK_BUFFER_SHORT;
	IP_CONTROL2 : IP_CONTROL2;
	IRTRANS_DECODE : IRTRANS_DECODE;
	IRTRANS_RCV_4 : IRTRANS_RCV_4;
	DRIVER_4 : DRIVER_4;
	IRTRANS_SERVER : IRTRANS_SERVER;
	IRTRANS_SND_8_1 : IRTRANS_SND_8;
	IRTRANS_SND_8_2 : IRTRANS_SND_8;
	Q0: BOOL;
	Q1: BOOL;
	Q2: BOOL;
	Q3: BOOL;
	error: BOOL;
	error_server: DWORD;
	Send_1_0: BOOL := TRUE;
	Send_1_1: BOOL;
	Send_1_2: BOOL;
	Send_1_3: BOOL;
	Send_1_4: BOOL;
	Send_1_5: BOOL;
	Send_1_6: BOOL;
	Send_1_7: BOOL;
	Send_2_0: BOOL := TRUE;
	Send_2_1: BOOL;
	Send_2_2: BOOL;
	Send_2_3: BOOL;
	Send_2_4: BOOL;
	Send_2_5: BOOL;
	Send_2_6: BOOL;
	Send_2_7: BOOL;
	R_ENABLE: BOOL;
	S_ENABLE: BOOL;
	MODE: BOOL := FALSE;
	KEY_1: BYTE;
	KEY_2: BYTE;
END_VAR
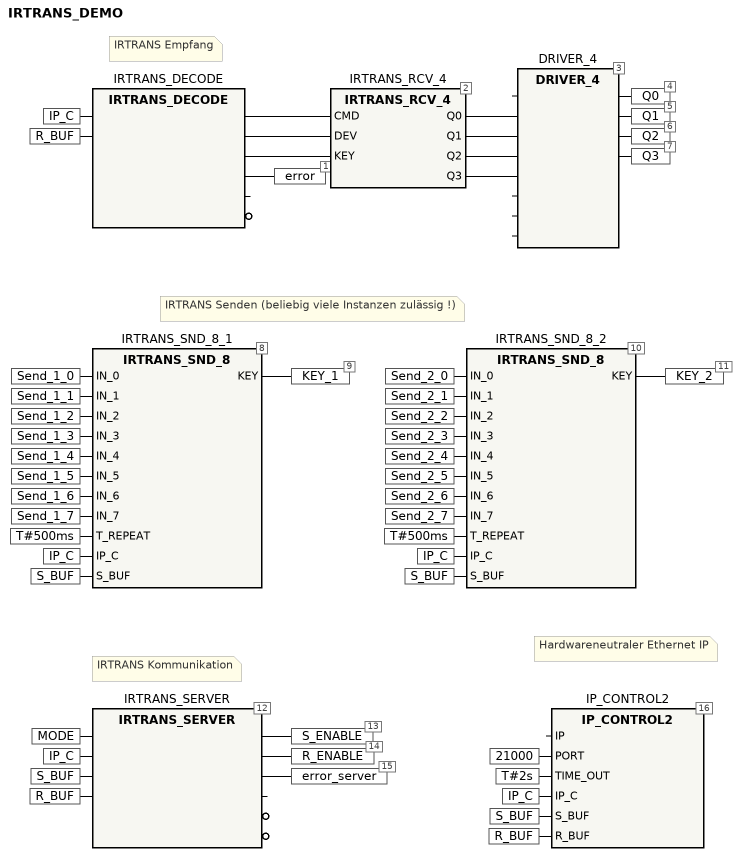
_CFC_ (* Continuous Function Chart, elements in execution order *)
(* IRTRANS Senden (beliebig viele Instanzen zulässig !) *)
(* IRTRANS Kommunikation *)
(* IRTRANS Empfang *)
(* Hardwareneutraler Ethernet IP *)
#0 IRTRANS_DECODE:IRTRANS_DECODE(IP_C, R_BUF)
#1 error <= #0.out 4
#2 IRTRANS_RCV_4:IRTRANS_RCV_4(CMD: #0.out 1, DEV: #0.out 2, KEY: #0.out 3)
#3 DRIVER_4:DRIVER_4(-, #2.Q0, #2.Q1, #2.Q2, #2.Q3, -, -, -, Toggle_Mode := TRUE)
#4 Q0 <= #3.out 1
#5 Q1 <= #3.out 2
#6 Q2 <= #3.out 3
#7 Q3 <= #3.out 4
#8 IRTRANS_SND_8_1:IRTRANS_SND_8(IN_0: Send_1_0, IN_1: Send_1_1, IN_2: Send_1_2, IN_3: Send_1_3, IN_4: Send_1_4, IN_5: Send_1_5, IN_6: Send_1_6, IN_7: Send_1_7, T_REPEAT: T#500ms, IP_C: IP_C, S_BUF: S_BUF)
#9 KEY_1 <= #8.KEY
#10 IRTRANS_SND_8_2:IRTRANS_SND_8(IN_0: Send_2_0, IN_1: Send_2_1, IN_2: Send_2_2, IN_3: Send_2_3, IN_4: Send_2_4, IN_5: Send_2_5, IN_6: Send_2_6, IN_7: Send_2_7, T_REPEAT: T#500ms, IP_C: IP_C, S_BUF: S_BUF)
#11 KEY_2 <= #10.KEY
#12 IRTRANS_SERVER:IRTRANS_SERVER(MODE, IP_C, S_BUF, R_BUF)
#13 S_ENABLE <= #12.out 1
#14 R_ENABLE <= #12.out 2
#15 error_server <= #12.out 3
#16 IP_CONTROL2:IP_CONTROL2(IP: -, PORT: 21000, TIME_OUT: T#2s, IP_C: IP_C, S_BUF: S_BUF, R_BUF: R_BUF)
_END_CFC_
END_PROGRAM

(* POU IP_CONTROL2, ST *)
FUNCTION_BLOCK IP_CONTROL2
VAR_IN_OUT
	IP_C : IP_C; (* IP_Control Verwaltungsstruktur *)
	S_BUF : NETWORK_BUFFER_SHORT; (* Externer Sendbuffer *)
	R_BUF : NETWORK_BUFFER_SHORT; (* Externer Receivebuffer *)
END_VAR
VAR_INPUT
	IP : DWORD; (* IP Adresse *)
	PORT : WORD; (* Port Nummer *)
	TIME_OUT : TIME; (* Ueberwachungszeit Connect / Send / Receive *)
END_VAR
VAR
	c_time : UDINT; (* CONNECT-Time (Zeit bei nicht vorhandener Verbindung) *)
	s_time : UDINT; (* SEND-Time    (Zeit seit letzten Datensenden) *)
	r_time : UDINT; (* RECEIVE-Time (Zeit seit letztem Datenempfang) *)

	c_enable : BOOL; (* Connect: freigabe *)
	c_ip : DWORD; (* Connect: aktuelle IP-Adresse *)
	c_port : WORD; (* Connect: aktuelle Port-Nummer *)
	c_mode : BYTE; (* Connect: aktueller Mode UDP/TCP...... *)
	c_status : BYTE; (* Connect: Status (Errorcode) *)
	c_ready : BOOL; (* Connect: Verbindung aufgebaut *)
	c_ready_old : BOOL; (* Connect: letzter Zustand von c_ready für Flankenauswertung *)
	c_select : BOOL; (* non blocking mode - abfrage über select durchführen *)
	c_fdWrite : SOCKET_FD_SET;
	c_Timeout : SOCKET_TIMEVAL;

	s_total : INT; (* Send: Gesamtanzahl Bytes zum senden *)
	s_cur_pos : INT; (* Send: aktuelle Sendeposition *)
	s_cur_size : INT; (* Send: aktuelle Sendegroesse *)
	s_max_size : INT; (* Send: maximale Telegrammlänge fuer Senden *)
	s_start : BOOL; (* Send: Sende modus aktivieren *)
	s_active : BOOL; (* Send: Daten senden ist aktiv *)
	s_req : BOOL; (* Send: Start Daten senden *)
	s_done : BOOL; (* Send: ohne Fehler beendet *)
	s_status : BYTE; (* Send: Status (Errorcodes) *)

	r_status : BYTE; (* Receive: Status (Errorcodes) *)
	r_count : INT; (* Receive: Anzahl empfangener Bytes *)
	r_offset : INT; (* Receive: aktuelle Position in externen Receivebuffer *)
	r_max_size : INT; (* Receive: groesse des externen Empfangbuffers*)

	new_connection : BOOL; (* Neue Verbindungsparameter vorhanden *)
	tx : DWORD; (* letzter zeitwert *)
	error_time : DWORD; (* aktueller Timeout-Wert *)

	state: BYTE; (* schrittmerker für connect *)
	server_socket : DINT:= SOCKET_INVALID;
	socket : DINT:= SOCKET_INVALID;
	sockaddr : SOCKADDRESS;
	sockaddr_size : DWORD;
	plc_841 : BOOL;
	dint_true : DINT := 1;
	bytes_received : DINT;
	bytes_sent : DINT;
	udp_mode : BOOL;

	(*LOG_MSG : LOG_MSG;
	_debug_enable : BOOL := TRUE;
	debug_index : INT;
	debug_ID : INT;
	debug_lasterror : DWORD;
	debug_last_id : INT := 255;
	state_last: BYTE;*)

END_VAR

VAR CONSTANT
	STOP : BYTE := 0;
	TS_INIT: BYTE := 1;
	TS_OPEN : BYTE:= 2;
	UDP_INIT : BYTE:= 31;
	TC_INIT : BYTE:= 51;
	TC_CONNECT : BYTE:= 52;
	C_WAIT : BYTE:= 250;
	C_CLOSE : BYTE:= 251;
END_VAR

(*

version 1.5		10. nov. 2010
programmer 		ks
tested by			ks

IP_CONTROL ist ein Wrapper-Baustein um eine Hersteller neutrale Schnittstelle zum Ethernet zu schaffen
*)
(* ---------------------- Debug-Message ----------------------------*)
(*IF _debug_enable THEN
	IF IP_C.FIFO.ID > BYTE#0 THEN (* nur wenn Teilnehmer ID's vorhanden sind *)
		debug_index := IP_C.FIFO.NR;
		debug_ID := BYTE_TO_INT(IP_C.FIFO.X[debug_index]);
	END_IF;
END_IF;*)
(* -----------------------------------------------------------------------------*)

(* read system time *)
tx := T_PLC_MS();

IF IP_C.C_PORT = 0 THEN
	IP_C.C_PORT := PORT; (* uebergebenen PORT durch parametrierten PORT ersetzen *)
END_IF;
IF IP_C.C_IP = 0 AND IP_C.C_MODE < 4 THEN
	IP_C.C_IP := IP; (* uebergebene IP durch paramtrierte IP ersetzen *)
END_IF;

new_connection := c_ip <> IP_C.C_IP OR c_mode <> IP_C.C_MODE OR c_port <> IP_C.C_PORT; (* neue Verbindungs erwünscht ? *)
c_enable := IP_C.C_ENABLE AND NOT new_connection;

IF IP_C.C_ENABLE AND IP_C.ERROR = 0 AND state = STOP THEN (* Freigabe,kein Fehler,kein Socket offen *)
	c_ip   := IP_C.C_IP;
	c_mode := IP_C.C_MODE;
	c_port := IP_C.C_PORT;
	plc_841 := ADR(%MW0)=16#30000000; (*750-841*)
	udp_mode := C_MODE.0; (* Mode 1,3,5 = udp *)

	error_time := TIME_TO_DWORD(MAX(T#200ms,TIME_OUT));
	IP_C.TIME_RESET := TRUE; (* Alle Timer ruecksetzen *)

	r_max_size := SIZEOF(R_BUF.BUFFER);
	s_max_size := SIZEOF(S_BUF.BUFFER);

	IF C_MODE.0 THEN (* Mode: 1,3,5 = UDP CLIENT/SERVER *)
		state := UDP_INIT;
	ELSIF C_MODE = 0 THEN (* Mode: 0 = TCP CLIENT *)
		state := TC_INIT;
	ELSE
		state := TS_INIT; (* Mode: 2,4 = TCP SERVER *)
	END_IF;

	(* ---------------------- Debug-Message ----------------------------*)
	(*IF _debug_enable THEN
		LOG_CL.NEW_MSG := 'IP_CON: MODE ~1 / IP ~2 / PORT ~3 /ID ~6';
		LOG_CL.PRINTF[1] := BYTE_TO_STRING(C_MODE);
		LOG_CL.PRINTF[2] := IP4_TO_STRING(c_ip);
		LOG_CL.PRINTF[3] := WORD_TO_STRING(c_port);
		LOG_CL.PRINTF[6] := INT_TO_STRING(debug_ID);
		LOG_MSG();
	END_IF;*)
	(* -----------------------------------------------------------------------------*)

END_IF;

(* ---------------------- Debug-Message ----------------------------*)
(*IF  _debug_enable THEN
	IF state <> state_last THEN
		LOG_CL.NEW_MSG := 'IP_STEP ~1 -IP_ID ~6';
		LOG_CL.PRINTF[1] := BYTE_TO_STRING(state);
		LOG_CL.PRINTF[6] := INT_TO_STRING(debug_ID);
		LOG_MSG();
		state_last := state;
	END_IF;
END_IF;*)
(* -----------------------------------------------------------------------------*)

(* ---------------------------------------------- *)

CASE state OF

UDP_INIT: (* UDP_CLIENT + SERVER *)
	socket := SysSockCreate(SOCKET_AF_INET, SOCKET_DGRAM, SOCKET_IPPROTO_UDP);
	IF socket < 0 THEN
		c_status := 1; (* SysSockCreate failed *)
		state := C_CLOSE;
	ELSE
		SysSockSetOption(socket, SOCKET_SOL, SOCKET_SO_BROADCAST, ADR(dint_true), SIZEOF(dint_true)); (* allow broadcast *)
		SysSockIoctl(socket, SOCKET_FIONBIO, ADR(dint_true)); (* put socket in non-blocking mode *)
		sockaddr.sin_family := SOCKET_AF_INET;
		sockaddr.sin_port := SysSockHtons(c_port);
		sockaddr.sin_addr := SEL(c_mode = 1, SOCKET_INADDR_ANY, SysSockNtohl(c_ip));

		IF c_mode >= 2 THEN (* SERVER Mode *)
			IF SysSockBind(socket, ADR(sockaddr), SIZEOF(sockaddr)) THEN
				c_ready := TRUE; (* Connected *)
				state:= C_WAIT;
			ELSE
				c_status := 2; (* SysSockBind failed *)
				state := C_CLOSE;
			END_IF;
		ELSE
			c_ready := TRUE; (* Connected *)
			state:= C_WAIT;
		END_IF;
	END_IF;

(* ---------------------------------------------- *)

TC_INIT: (* TCP-CLIENT (AKTIV) *)
	socket := SysSockCreate(SOCKET_AF_INET, SOCKET_STREAM, SOCKET_IPPROTO_TCP);
	IF socket < 0 THEN
		c_status := 1;  (* SysSockCreate failed *)
		state := C_CLOSE;
	ELSE
		IF plc_841 THEN
			SysSockSetOption(socket,6,SOCKET_TCP_NODELAY, ADR(dint_true), SIZEOF(dint_true)); (* Set Push-Bit *)
		END_IF;
		SysSockIoctl(socket, SOCKET_FIONBIO, ADR(dint_true)); (* NonBlocking mode *)
		sockaddr.sin_family := SOCKET_AF_INET;
		sockaddr.sin_port := SysSockNtohs(c_port);
		sockaddr.sin_addr := SysSockNtohl(c_ip);
		c_select := FALSE;
		state := TC_CONNECT;
	END_IF;

(* ---------------------------------------------- *)

TC_CONNECT:
	IF NOT c_enable OR c_status = 255 THEN (* keine freigabe oder connect timeout *)
			state:= C_CLOSE;
	ELSE
		IF c_select = FALSE THEN
			IF SysSockConnect(socket,ADR(sockaddr),SIZEOF(sockaddr)) THEN
				c_ready := TRUE; (* Connected *)
				state:= C_WAIT;
			ELSE
				c_select := TRUE; (* Connect durchgeführt, aber noch nicht verbunden, dann mit select-abfrage weitermachen *)
			END_IF;
		ELSE
			c_Timeout.tv_sec := 0;
			c_Timeout.tv_usec := 0;
			c_fdWrite.fd_count := 1;
			c_fdWrite.fd_array[0] := socket;
			IF SysSockSelect(SOCKET_FD_SETSIZE,0,ADR(c_fdWrite),0, ADR(c_Timeout)) > 0 THEN
				c_ready := TRUE; (* Connected *)
				state:= C_WAIT;
			END_IF;
		END_IF;
	END_IF;

(* ---------------------------------------------- *)

TS_INIT: (* TCP-SERVER (PASSIV) *)
	server_socket := SysSockCreate(SOCKET_AF_INET, SOCKET_STREAM, SOCKET_IPPROTO_IP); (* Create Socket *)
	IF server_socket = SOCKET_INVALID THEN
		c_status := 1; (* SysSockCreate failed *)
		state:= C_CLOSE;
	ELSE (* Address bindings *)
		sockaddr.sin_family:= SOCKET_AF_INET;
		sockaddr.sin_port := SysSockHtons(c_port);
		sockaddr.sin_addr := SOCKET_INADDR_ANY;
		IF NOT SysSockBind(server_socket, ADR(sockaddr), SIZEOF(sockaddr)) THEN
			c_status := 2; (* SysSockBind failed *)
			state := C_CLOSE;
		ELSIF NOT SysSockListen(server_socket, 1) THEN (* erzeugt Warteschlange für eine Verbindung *)
			c_status := 3; (* SysSockListen failed *)
			state:= C_CLOSE;
		ELSE
			SysSockIoctl(server_socket, SOCKET_FIONBIO, ADR(dint_true)); (* NonBlocking mode *)
			state:= TS_OPEN;
		END_IF;
	END_IF;

(* ---------------------------------------------- *)

TS_OPEN: (* Waiting for incomming connection *)
	sockaddr_size := SIZEOF(sockaddr);
	socket := SysSockAccept(server_socket, ADR(sockaddr), ADR(sockaddr_size));

	IF socket <> SOCKET_INVALID THEN (* neuer Verbindungswunsch vorhanden *)
		IF c_mode = BYTE#2 AND sockaddr.sin_addr <> SysSockNtohl(c_ip) THEN (* Mode 2 = TCP + PASSIVE + PORT + IP  auf richtige Partner-IP prüfen *)
			state:= C_CLOSE;
		ELSE
			IF plc_841 THEN
				SysSockSetOption(socket, 6, SOCKET_TCP_NODELAY, ADR(dint_true), SIZEOF(dint_true)); (* Set Push-Bit *)
			END_IF;
			SysSockIoctl(socket, SOCKET_FIONBIO, ADR(dint_true)); (* NonBlocking mode *)
			c_ready := TRUE; (* Connected *)
			state := C_WAIT;
		END_IF;
	ELSIF NOT c_enable THEN (* keine freigabe mehr ? *)
			state:= C_CLOSE;
	END_IF;

(* ---------------------------------------------- *)

C_WAIT: (* Warten auf Anforderung für Beenden *)
	IF NOT c_enable OR NOT c_ready THEN
		state:= C_CLOSE;
	END_IF

(* ---------------------------------------------- *)

C_CLOSE: (* Close the Sockets *)
	c_ready := FALSE;
	IF socket >= 0 THEN
		IF NOT plc_841 THEN SysSockShutdown(socket, 0); END_IF; (* 870 *)
		SysSockClose(socket);
		socket := SOCKET_INVALID;
	END_IF
	IF server_socket >= 0 THEN
		IF NOT plc_841 THEN SysSockShutdown(server_socket, 0); END_IF; (* 870 *)
		SysSockClose(server_socket);
		server_socket := SOCKET_INVALID;
	END_IF
	state:= STOP;
END_CASE;

(* ---------------------------------------------- *)

IF c_ready THEN
	IF NOT c_ready_old THEN (* Verbindung aufgebaut - positive Flanke erkannt *)
		IP_C.C_STATE := 254;
		IP_C.TIME_RESET := TRUE; (* Alle Timer ruecksetzen *)
		(* ---------------------- Debug-Message ----------------------------*)
		(*IF _debug_enable THEN
			LOG_CL.NEW_MSG := 'IP_CON: CONNECTED -IP_ID ~6';
			LOG_CL.PRINTF[6] := INT_TO_STRING(debug_ID);
			LOG_MSG();
		END_IF;*)
		(* -----------------------------------------------------------------------------*)
	ELSE
		IP_C.C_STATE := 255; (* Verbindung ist aufgebaut *)
	END_IF;
ELSE
	IF c_ready_old THEN (* Verbindung abgebaut - negative Flanke erkannt *)
		IP_C.C_STATE := 1;
		IP_C.MAILBOX[1] := 0; (* Receive Info rücksetzen *)
		IP_C.MAILBOX[2] := 0; (* Send-Pause rücksetzen *)
		IP_C.MAILBOX[3] := 0; (* Receive-Pause rücksetzen *)
		IF NOT new_connection THEN
			s_active := FALSE; (* Sendeaktivitäten stoppen *)
			s_req := FALSE; (* Sendefreigabe rücksetzen *)
			S_BUF.SIZE := 0; (* Sendelänge löschen *)
			IP_C.C_ENABLE := FALSE;
			IP_C.TIME_RESET := TRUE; (* Alle Timer ruecksetzen *)
		END_IF;
		(* ---------------------- Debug-Message ----------------------------*)
		(*IF _debug_enable THEN
			LOG_CL.NEW_MSG := 'IP_CON: DISCONNECTED';
			LOG_MSG();
		END_IF;*)
		(* -----------------------------------------------------------------------------*)
	ELSE
		IP_C.C_STATE := 0; (* Verbindung ist abgebaut *)
	END_IF;
END_IF;

c_ready_old := c_ready;

(* Der Datenempfang wird angehalten solange ein Sendevorgang läuft *)
(* sonst kann es vorkommen das die Antwort-daten schon empfangen werden, *)
(* bevor der Sendevorgang vom programm abgeschlossen wurde *)

IF c_ready AND NOT s_active AND IP_C.MAILBOX[3] = 0 THEN
	IF R_BUF.SIZE >= INT_TO_UINT(r_max_size) THEN
		R_BUF.SIZE := UINT#0;
		r_status := 254; (* Empfangsbuffer wegen Überlauf rückgesetzt *)
	END_IF;

	r_offset := SEL(udp_mode,UINT_TO_INT(R_BUF.SIZE),0);
	r_count := r_max_size - r_offset;

	IF udp_mode THEN
		bytes_received := SysSockRecvFrom(socket, ADR(R_BUF.BUFFER), r_count, 0, ADR(sockaddr), SIZEOF(sockaddr));

		IF c_mode = BYTE#3 AND sockaddr.sin_addr <> SysSockNtohl(c_ip) THEN (* Mode 3 = UDP + PASSIVE + PORT + IP  auf richtige Partner-IP prüfen *)
			bytes_received := 0;
			R_BUF.SIZE := UINT#0;
			sockaddr.sin_port := SysSockNtohs(c_port);
			sockaddr.sin_addr := SysSockNtohl(c_ip);
		END_IF;

	ELSE
		bytes_received := SysSockRecv(socket, ADR(R_BUF.BUFFER[r_offset]), r_count, 0);
	END_IF;

	(*UDP: IPC returns -1 if no data available or error occured,841 returns -1 if error occured and 0 if no data available*)
	CASE bytes_received OF
	-1: ; (* No data available or error occured *)
	 0: IF NOT udp_mode THEN (* TCP-Mode: socket wurde von remote geschlossen *)
			c_ready := FALSE;
		END_IF;
	ELSE (* daten wurden empfangen *)
  		r_time := tx; (* Receive Timer ruecksetzen *)
		R_BUF.SIZE := INT_TO_UINT(r_offset + DINT_TO_UINT(bytes_received)); (* aktuelle buffersize eintragen *)
		IP_C.MAILBOX[1] := IP_C.MAILBOX[1] + 1; (* Receive Info *)
		IF IP_C.MAILBOX[1] = 0 THEN IP_C.MAILBOX[1] := 1; END_IF;

		(* ---------------------- Debug-Message ----------------------------*)
		(*IF _debug_enable THEN
			LOG_CL.NEW_MSG := 'IP_REC DATA: POS: ~1 : SIZE: ~2 TOTAL ~3 -IP_ID ~6';
			LOG_CL.PRINTF[1] := INT_TO_STRING(r_offset);
			LOG_CL.PRINTF[2] := INT_TO_STRING(r_count);
			LOG_CL.PRINTF[3] := UINT_TO_STRING(R_BUF.SIZE);
			LOG_CL.PRINTF[6] := INT_TO_STRING(debug_ID);
			LOG_MSG();
		END_IF;*)
		(* -----------------------------------------------------------------------------*)

	END_CASE
END_IF;

(* ---------------------------------------------- *)

IF S_BUF.SIZE > 0 THEN
	IF c_ready AND c_enable THEN
		IF NOT s_active AND IP_C.MAILBOX[2] = 0 THEN
			(* Gesamtanzahl an Bytes limitieren und uebergeben *)
			s_total := LIMIT(0,UINT_TO_INT(S_BUF.SIZE),r_max_size);
			s_cur_pos  := 0;
			s_cur_size := 0;
			s_start := TRUE; (* Daten kopieren und senden anstossen *)
			s_active := TRUE; (* Sende-Betrieb aktivieren *)
			(* ---------------------- Debug-Message ----------------------------*)
			(*IF _debug_enable THEN
				LOG_CL.NEW_MSG := 'IP_SEN INIT: TOTAL: ~1 -IP_ID ~6';
				LOG_CL.PRINTF[1] := INT_TO_STRING(S_TOTAL);
				LOG_CL.PRINTF[6] := INT_TO_STRING(debug_ID);
				LOG_MSG();
			END_IF;*)
			(* -----------------------------------------------------------------------------*)
		END_IF;

		IF s_done OR s_start THEN (* Daten senden aktiv *)

			s_start := FALSE;
			s_cur_pos := s_cur_pos + s_cur_size; (* neue Sende-Datenposition bestimmen *)
			IF s_total > s_cur_pos THEN (* weitere Daten zum senden vorhanden ? *)
				s_cur_size := s_total - s_cur_pos;
				s_cur_size := LIMIT(0, s_cur_size, s_max_size); (* Telegrammlänge begrenzen *)

				(* ---------------------- Debug-Message ----------------------------*)
				(*IF _debug_enable THEN
					LOG_CL.NEW_MSG := 'IP_SEN DATA: POS: ~1 : SIZE: ~2 TOTAL ~3 -IP_ID ~6';
					LOG_CL.PRINTF[1] := INT_TO_STRING(S_CUR_POS);
					LOG_CL.PRINTF[2] := INT_TO_STRING(S_CUR_SIZE);
					LOG_CL.PRINTF[3] := INT_TO_STRING(S_TOTAL);
					LOG_CL.PRINTF[6] := INT_TO_STRING(debug_ID);
					LOG_MSG();
				END_IF;*)
				(* -----------------------------------------------------------------------------*)

				s_time := tx; (* Send Timer ruecksetzen *)
				s_req := TRUE;

			ELSE
				(* keine weitere Sendedaten vorhanden -> Senden beenden *)
				s_req := FALSE;
				s_active := FALSE;
				S_BUF.SIZE := 0;
				(* ---------------------- Debug-Message ----------------------------*)
				(*IF _debug_enable THEN
					LOG_CL.NEW_MSG := 'IP_SEN FINISH -IP_ID ~6';
					LOG_CL.PRINTF[6] := INT_TO_STRING(debug_ID);
					LOG_MSG();
				END_IF;*)
				(* -----------------------------------------------------------------------------*)
			END_IF;
		END_IF;
	END_IF;
END_IF;

IF s_req THEN
	s_done := FALSE;
	IF udp_mode THEN
		bytes_sent := SysSockSendTo(socket, ADR(S_BUF.BUFFER[s_cur_pos]), s_cur_size, 0, ADR(sockaddr), SIZEOF(sockaddr));
	ELSE
		bytes_sent := SysSockSend(socket, ADR(S_BUF.BUFFER[s_cur_pos]), s_cur_size, 0);
	END_IF;

	CASE bytes_sent OF
	-1:	; (* ERROR: Noch nicht bereit um Daten aufzunehmen -> nächsten Zyklus wieder probieren *)
	 0: IF NOT udp_mode THEN (* TCP-Mode: socket wurde von remote geschlossen *)
			c_ready := FALSE;
		END_IF;
	ELSE
		s_done := TRUE;
		s_cur_size := DINT_TO_INT(bytes_sent); (* Anzahl der wirklich versendeten Bytes übernehmen *)
		(* ---------------------- Debug-Message ----------------------------*)
		(*IF _debug_enable THEN
			LOG_CL.NEW_MSG := 'IP_SEN SEND_COUNT ~1 -IP_ID ~6';
			LOG_CL.PRINTF[1] := DINT_TO_STRING(s_cur_size);
			LOG_CL.PRINTF[6] := INT_TO_STRING(debug_ID);
			LOG_MSG();
		END_IF;*)
		(* -----------------------------------------------------------------------------*)
	END_CASE
END_IF;

(* ---------------------------------------------- *)

IF IP_C.TIME_RESET THEN (* Alle Timer ruecksetzen *)
	IP_C.TIME_RESET := FALSE; (* Reset rücksetzen *)
	c_time := tx; (* Connect Timer ruecksetzen *)
	s_time := tx; (* Send Timer ruecksetzen *)
	r_time := tx; (* Receive Timer ruecksetzen *)

	c_status := BYTE#0; (* letzten Connect Fehler rücksetzen *)
	s_status := BYTE#0; (* letzten Send Fehler rücksetzen *)
	r_status := BYTE#0; (* letzten Receive Fehler rücksetzen *)
END_IF;

IF c_status = 0 AND tx - c_time > error_time AND c_enable AND NOT c_ready AND c_mode < 2 THEN (* Connect Timeout *)
	c_status := 255; (* Timeout-Fehler ausgeben *)
END_IF;
IF s_status = 0 AND tx - s_time > error_time AND s_active THEN (* Send Timeout *)
	s_status := 255; (* Timeout-Fehler ausgeben *)
END_IF;
IF r_status = 0 AND tx - r_time > error_time AND c_ready AND IP_C.R_OBSERVE THEN (* Receive Timeout *)
	r_status := 255; (* Timeout-Fehler ausgeben *)
END_IF;

IP_C.ERROR := DWORD_OF_BYTE(c_status,s_status,r_status,0);

(* ---------------------- Debug-Message ----------------------------*)
(*IF  _debug_enable THEN
	IF (IP_C.ERROR <> debug_lasterror) THEN
		LOG_CL.NEW_MSG := 'IP_ERROR ~1 -IP_ID ~6';
		LOG_CL.PRINTF[1] := DWORD_TO_STRING(IP_C.ERROR);
		LOG_CL.PRINTF[6] := INT_TO_STRING(debug_ID);
		LOG_MSG();

		debug_lasterror := IP_C.ERROR;
		debug_last_id := debug_ID;
	END_IF;
END_IF;*)
(* -----------------------------------------------------------------------------*)

(* revision history
ks	18. oct. 2008	rev 1.0
	original version
ks	05. jan. 2009	rev 1.1
	zusätzlichen Parameter "Port" hinzugefügt, und Code bei Verbindungsaufbau angepasst
ks	28. feb. 2009	rev 1.2
	connect code angepasst und verkürzung der zyklen bei Send
ks	20. oct. 2009	rev 1.3
	network_buffer basis 0
ks	06. dec. 2009	rev 1.4
	receive_count MAILBOX[1]
ks	10. nov. 2010	rev 1.5
	send_pause MAILBOX[2] and receive_pause MAILBOX[3] 
*)
END_FUNCTION_BLOCK

(* POU IRTRANS_DECODE, ST *)
FUNCTION_BLOCK IRTRANS_DECODE
VAR_IN_OUT
	IP_C : IP_C; (* IP_Control Verwaltungsstruktur *)
	R_BUF : NETWORK_BUFFER_SHORT;
END_VAR
VAR_OUTPUT
	CMD : BOOL;
	DEV : STRING;
	KEY : STRING;
	ERROR : BOOL;
END_VAR
VAR
	i : INT;
	stop : INT;
	pt : POINTER TO BYTE;
	buffer : POINTER TO ARRAY[0..32000] OF BYTE;
	size : UINT;
	z : BYTE;
END_VAR

(*

version 1.2		06. dec. 2009
programmer 		ks
tested by		ks

*)
size := R_BUF.SIZE;

(* do nothing if the buffer is empty *)
IF size > 0 AND IP_C.MAILBOX[1] <> z THEN
	i := 0;
	error := TRUE;
	stop := size - 2;
	(* read characters before first comma and store in device *)
	pt := ADR(dev);
	buffer := ADR(R_BUF.BUFFER);
	WHILE i < stop DO
		IF buffer^[i] = 44 THEN EXIT; END_IF;
		pt^ := buffer^[i];
		pt := pt + 1;
		i := i + 1;
	END_WHILE;
	(* terminate the device string *)
	pt^ := 0;
	(* read after first comma and store in key *)
	i := i + 1;
	pt := ADR(key);
	WHILE i < stop DO
		pt^ := buffer^[i];
		pt := pt + 1;
		i := i + 1;
	END_WHILE;
	(* terminate the key string *)
	pt^:= 0;
	(* check if last two characters are $R$N 13, 10 *)
	IF buffer^[i] <> 13 AND buffer^[i+1] <> 10 THEN	RETURN;	END_IF;
	(* check if device and key are present *)
	IF LEN(dev) = 0 OR LEN(key) = 0 THEN RETURN; END_IF;
	(* a valid transmission has been received *)
	cmd := TRUE;
	error := FALSE;
ELSE
	error := FALSE;
	cmd := FALSE;
END_IF;

z := IP_C.MAILBOX[1];

(* revision history
ks	18. oct. 2008	rev 1.0
	original version
ks	20. oct. 2009	rev 1.1
	Networkbuffer und Buffer-funktionen auf Basis 0
ks	06. dec. 2009	rev 1.2
	Codeanpassung für IRTRANS_SERVER
*)
END_FUNCTION_BLOCK

(* POU IRTRANS_RCV_4, ST *)
FUNCTION_BLOCK IRTRANS_RCV_4
VAR_INPUT CONSTANT
	DEV_CODE : STRING;
	KEY_CODE_0 : STRING;
	KEY_CODE_1 : STRING;
	KEY_CODE_2 : STRING;
	KEY_CODE_3 : STRING;
END_VAR
VAR_INPUT
	CMD : BOOL;
END_VAR
VAR_IN_OUT
	DEV : STRING;
	KEY : STRING;
END_VAR
VAR_OUTPUT
	Q0, Q1, Q2, Q3 : BOOL;
END_VAR
VAR_TEMP
	decode: BOOL;
END_VAR

(*

version 1.3	06. dec. 2009
programmer 	hugo
tested BY	oscat

*)
decode := cmd AND dev_code = dev;

Q0 := key = key_code_0 AND decode;
Q1 := key = key_code_1 AND decode;
Q2 := key = key_code_2 AND decode;
Q3 := key = key_code_3 AND decode;



(* revision history
hm	2. jan 2008		rev 1.0
	original version

hm	17. oct. 2008	rev 1.1
	improved performance

hm	19. oct. 2008	rev 1.2
	changed input device_code to dev_code and device to dev for compatibility reasons

hm	06. dec. 2008	rev 1.3
	IRTRANS_1 renamed to IRTRANS_RCV_4

*)
END_FUNCTION_BLOCK

(* POU IRTRANS_SERVER, ST *)
FUNCTION_BLOCK IRTRANS_SERVER
VAR_IN_OUT
	IP_C : IP_C; (* IP_Control Verwaltungsstruktur *)
	S_BUF : NETWORK_BUFFER_SHORT;
	R_BUF : NETWORK_BUFFER_SHORT;
END_VAR
VAR_INPUT
	UDP_TCP : BOOL;
END_VAR
VAR_OUTPUT
	S_ENABLE : BOOL;
	R_ENABLE : BOOL;
	ERROR : DWORD;
END_VAR
VAR
	t : TON;
END_VAR

(*
version 1.0		06. dec. 2009
programmer 		ks
tested by		ks
*)
IF NOT IP_C.C_ENABLE THEN
	(* IP Datenverkehr einrichten *)
	IP_C.C_PORT := WORD#0; (* Portnummer eintragen *)
	IP_C.C_IP := DWORD#00; (* IP eintragen *)
	IP_C.C_MODE := SEL(UDP_TCP,5,4); (* 4 = Mode: TCP+PASSIV+PORT / 5 = Mode: UDP+PASSIV+PORT*)
	IP_C.C_ENABLE := TRUE; (* Verbindungsaufbau freigeben *)
	IP_C.R_OBSERVE := FALSE; (* Datenempfang ueberwachen *)
	IP_C.TIME_RESET := TRUE; (* Zeitueberwachung rücksetzen *)
	S_BUF.SIZE := UINT#0; (* Sendedaten rücksetzen *)
END_IF;

R_ENABLE := IP_C.C_STATE > 127;
S_ENABLE := R_ENABLE AND (IP_C.MAILBOX[1] > 0 OR IP_C.C_MODE <> 5);

t(IN:= IP_C.ERROR > 0, PT:=T#5s);
IF t.Q THEN
	IP_C.TIME_RESET := TRUE; (* Error Reset *)
END_IF;

(* revision history
hm	6. dec 2009		rev 1.0
	original version
*)
END_FUNCTION_BLOCK

(* POU IRTRANS_SND_8, ST *)
FUNCTION_BLOCK IRTRANS_SND_8
VAR_INPUT CONSTANT
	DEV_CODE : STRING;
	KEY_CODE_0 : STRING;
	KEY_CODE_1 : STRING;
	KEY_CODE_2 : STRING;
	KEY_CODE_3 : STRING;
	KEY_CODE_4 : STRING;
	KEY_CODE_5 : STRING;
	KEY_CODE_6 : STRING;
	KEY_CODE_7 : STRING;
END_VAR
VAR_INPUT
	IN_0 : BOOL;
	IN_1 : BOOL;
	IN_2 : BOOL;
	IN_3 : BOOL;
	IN_4 : BOOL;
	IN_5 : BOOL;
	IN_6 : BOOL;
	IN_7 : BOOL;
	T_REPEAT : TIME;
END_VAR
VAR_IN_OUT
	IP_C : IP_C; (* IP_Control Verwaltungsstruktur *)
	S_BUF : NETWORK_BUFFER_SHORT;
END_VAR
VAR_OUTPUT
	KEY : BYTE;
END_VAR
VAR
	skey : STRING;
	size : INT;
	str : STRING;
	t : TON;
	k : BYTE;
	lk : BYTE;
	d : BOOL;
END_VAR

(*
version 1.0		06. dec. 2009
programmer 		ks
tested by		ks
*)
d := IP_C.C_STATE > 127 AND (IP_C.MAILBOX[1] > 0 OR IP_C.C_MODE <> 5);
IF NOT d THEN RETURN; END_IF;

t(IN:= lk = k , PT:=T_REPEAT);

IF S_BUF.SIZE = 0 THEN
	IF IN_0 THEN
		skey := KEY_CODE_0; k := 1;
	ELSIF IN_1 THEN
		skey := KEY_CODE_1; k := 2;
	ELSIF IN_2 THEN
		skey := KEY_CODE_2; k := 3;
	ELSIF IN_3 THEN
		skey := KEY_CODE_3; k := 4;
	ELSIF IN_4 THEN
		skey := KEY_CODE_4; k := 5;
	ELSIF IN_5 THEN
		skey := KEY_CODE_5; k := 6;
	ELSIF IN_6 THEN
		skey := KEY_CODE_6; k := 7;
	ELSIF IN_7 THEN
		skey := KEY_CODE_7; k := 8;
	ELSE
		lk := 0;
		KEY := 0;
		RETURN; (* beenden wenn kein Key aktiv *)
	END_IF;

	IF lk <> k OR T.Q THEN (* anderer Key oder repeat wartezeit abgelaufen *)
		str := CONCAT('snd ',dev_code);
		str := CONCAT(str,',');
		str := CONCAT(str,skey);
		size := LEN(str);
		_STRING_TO_BUFFER(STR:=str, POS:=0, PT:=ADR(S_BUF.BUFFER), SIZE:=size);
		S_BUF.SIZE := size; (* Sendelänge eintragen *)
		KEY := k;
		lk := k; (* letzten Key speichern *)
		t(IN:=FALSE); (* Reset Time *)
	END_IF;
END_IF;

(* revision history
hm	6. dec 2009		rev 1.0
	original version
*)
END_FUNCTION_BLOCK

(* POU MB_CLIENT_DEMO, CFC *)
PROGRAM MB_CLIENT_DEMO
VAR
	IP_CONTROL2_1: IP_CONTROL2;
	MB_CLIENT_1: MB_CLIENT;
	IP_C: IP_C;
	S_BUF: NETWORK_BUFFER_SHORT;
	R_BUF: NETWORK_BUFFER_SHORT;
	DATA: ARRAY [0..255] OF WORD;
	W_DATA_BITPOS: INT;
	W_DATA_ADR: INT;
	W_POINTS: INT;
	W_ADDR: INT;
	R_DATA_BITPOS: INT;
	R_DATA_ADR: INT;
	R_POINTS: INT;
	R_ADDR: INT;
	FC: INT;
	ENABLE: BOOL;
END_VAR
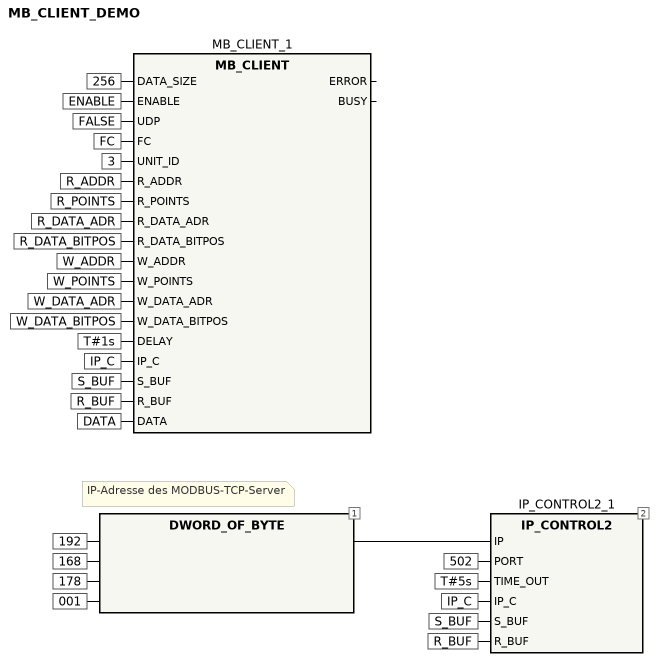
_CFC_ (* Continuous Function Chart, elements in execution order *)
(* IP-Adresse des MODBUS-TCP-Server *)
#0 MB_CLIENT_1:MB_CLIENT(DATA_SIZE: 256, ENABLE: ENABLE, UDP: FALSE, FC: FC, UNIT_ID: 3, R_ADDR: R_ADDR, R_POINTS: R_POINTS, R_DATA_ADR: R_DATA_ADR, R_DATA_BITPOS: R_DATA_BITPOS, W_ADDR: W_ADDR, W_POINTS: W_POINTS, W_DATA_ADR: W_DATA_ADR, W_DATA_BITPOS: W_DATA_BITPOS, DELAY: T#1s, IP_C: IP_C, S_BUF: S_BUF, R_BUF: R_BUF, DATA: DATA)
#1 DWORD_OF_BYTE(192, 168, 178, 001)
#2 IP_CONTROL2_1:IP_CONTROL2(IP: #1, PORT: 502, TIME_OUT: T#5s, IP_C: IP_C, S_BUF: S_BUF, R_BUF: R_BUF)
_END_CFC_
(* the same logic as Structured Text *)
(* IP-Adresse des MODBUS-TCP-Server *)
MB_CLIENT_1(DATA_SIZE := 256, ENABLE := ENABLE, UDP := FALSE, FC := FC, UNIT_ID := 3, R_ADDR := R_ADDR, R_POINTS := R_POINTS, R_DATA_ADR := R_DATA_ADR, R_DATA_BITPOS := R_DATA_BITPOS, W_ADDR := W_ADDR, W_POINTS := W_POINTS, W_DATA_ADR := W_DATA_ADR, W_DATA_BITPOS := W_DATA_BITPOS, DELAY := T#1s, IP_C := IP_C, S_BUF := S_BUF, R_BUF := R_BUF, DATA := DATA);
IP_CONTROL2_1(IP := DWORD_OF_BYTE(192, 168, 178, 001), PORT := 502, TIME_OUT := T#5s, IP_C := IP_C, S_BUF := S_BUF, R_BUF := R_BUF);
END_PROGRAM

(* POU MB_CLIENT, ST *)
FUNCTION_BLOCK MB_CLIENT
VAR_IN_OUT
	IP_C : IP_C;
	S_BUF : NETWORK_BUFFER_SHORT;
	R_BUF : NETWORK_BUFFER_SHORT;
	DATA : ARRAY [0..255] OF WORD;
END_VAR
VAR_INPUT
	DATA_SIZE : INT;
	ENABLE : BOOL;
	UDP : BOOL;
	FC : INT;
	UNIT_ID : BYTE;
	R_ADDR : INT;
	R_POINTS : INT;
	R_DATA_ADR : INT;
	R_DATA_BITPOS : INT;
	W_ADDR : INT;
	W_POINTS : INT;
	W_DATA_ADR : INT;
	W_DATA_BITPOS : INT;
	DELAY : TIME;
END_VAR
VAR_OUTPUT
	ERROR : DWORD;
	BUSY : BOOL;
END_VAR
VAR
	ip_state : BYTE;
	ip_id : BYTE;
	ip_fifo : ip_fifo;
	mask : DWORD;
	w_tmp : WORD;
	idx1 : INT;
	idx2 : INT;
	stop : INT;
	i : INT;
	bit_pos : INT;
	w_mask : WORD;
	b_mask : BYTE;
	count : INT;
	state : INT;
	transaction_id : INT;
	response : INT;
	comp : INT;
	ton_1 : TON;
END_VAR

(*
version 1.2		20. oct. 2009
programmer 		ks
tested BY		ks

MB_CLIENT ermöglicht das Lesen/Schreiben von Daten über das Protokoll Modbus over Ethernet (OpenModbus)
*)
CASE state OF

00: (* Warten auf Delay-Time *)
	TON_1(IN:=ENABLE,PT:=DELAY);

	IF TON_1.Q OR DELAY = T#0s THEN
		TON_1(IN:=FALSE);
		state := 20;
		IP_STATE := BYTE#1; (* Anmelden *)
	END_IF;

20: (* Bei IP_Control anmelden *)
	IF IP_STATE = BYTE#3 THEN
		(* IP Datenverkehr einrichten *)
		IP_C.C_PORT := WORD#0; (* Port von IP_CONTROL verwenden *)
		IP_C.C_IP := DWORD#0; (* IP von IP_CONTROL verwenden *)
		IP_C.C_MODE := BOOL_TO_BYTE(UDP); (* Mode: 0=TCP+ACTIVE+IP , 1=UDP+ACTIVE+IP *)
		IP_C.TIME_RESET := TRUE; (* Zeitueberwachung rücksetzen *)
		IP_C.C_ENABLE := TRUE; (* Verbindungsaufbau freigeben *)
		IP_C.R_OBSERVE := TRUE; (* Empfangsueberwachung *)
		ERROR := DWORD#00; (* letzten Fehler rücksetzen *)

